LIN {X 0,Y 485.565,Z 374.75,A -85,B 0,C 180,E1 23378.433,E2 23378.433} C_VEL
LIN {X 0,Y 487.506,Z 347.224,A -85,B 0,C 180,E1 23374.747,E2 23374.747} C_VEL
LIN {X 0,Y 489.864,Z 321.169,A -85,B 0,C 180,E1 23371.121,E2 23371.121} C_VEL
LIN {X 0,Y 489.847,Z 318.644,A -85,B 0,C 180,E1 23370.733,E2 23370.733} C_VEL
LIN {X 0,Y 486.96,Z 308.048,A -85,B 0,C 180,E1 23368.702,E2 23368.702} C_VEL
LIN {X 0,Y 483.664,Z 298.045,A -85,B 0,C 180,E1 23366.497,E2 23366.497} C_VEL
LIN {X 0,Y 480.889,Z 290.899,A -85,B 0,C 180,E1 23364.593,E2 23364.593} C_VEL
LIN {X 0,Y 480.887,Z 290.899,A -85,B 0,C 180,E1 23360.949,E2 23360.949} C_VEL
LIN {X 0,Y 480.886,Z 290.899,A -85,B 0,C 180,E1 23357.325,E2 23357.325} C_VEL
LIN {X 0,Y 480.891,Z 290.899,A -85,B 0,C 180,E1 23353.65,E2 23353.65} C_VEL
LIN {X 0,Y 480.897,Z 290.898,A -85,B 0,C 180,E1 23349.976,E2 23349.976} C_VEL
LIN {X 0,Y 480.854,Z 290.925,A -85,B 0,C 180,E1 23348.951,E2 23348.951} C_VEL
LIN {X 0,Y 482.165,Z 294.329,A -85,B 0,C 180,E1 23348.168,E2 23348.168} C_VEL
LIN {X 0,Y 482.997,Z 296.239,A -85,B 0,C 180,E1 23347.74,E2 23347.74} C_VEL
LIN {X 0,Y 486.121,Z 303.618,A -85,B 0,C 180,E1 23346.266,E2 23346.266} C_VEL
LIN {X 0,Y 489.9,Z 313.848,A -85,B 0,C 180,E1 23344.569,E2 23344.569} C_VEL
LIN {X 0,Y 492.294,Z 321.57,A -85,B 0,C 180,E1 23343.465,E2 23343.465} C_VEL
LIN {X 0,Y 489.453,Z 352.379,A -85,B 0,C 180,E1 23340.575,E2 23340.575} C_VEL
LIN {X 0,Y 487.08,Z 389.197,A -85,B 0,C 180,E1 23337.373,E2 23337.373} C_VEL
LIN {X 0,Y 488.749,Z 404.821,A -85,B 0,C 180,E1 23337.007,E2 23337.007} C_VEL
LIN {X 0,Y 487.087,Z 540.591,A -85,B 0,C 180,E1 23334.828,E2 23334.828} C_VEL
LIN {X 0,Y 486.559,Z 592.008,A -85,B 0,C 180,E1 23334.024,E2 23334.024} C_VEL
LIN {X 0,Y 485.998,Z 611.058,A -85,B 0,C 180,E1 23333.512,E2 23333.512} C_VEL
LIN {X 0,Y 485.301,Z 630.353,A -85,B 0,C 180,E1 23332.758,E2 23332.758} C_VEL
LIN {X 0,Y 484.52,Z 648.608,A -85,B 0,C 180,E1 23331.806,E2 23331.806} C_VEL
LIN {X 0,Y 483.712,Z 665.393,A -85,B 0,C 180,E1 23330.7,E2 23330.7} C_VEL
LIN {X 0,Y 482.923,Z 681.405,A -85,B 0,C 180,E1 23329.41,E2 23329.41} C_VEL
LIN {X 0,Y 482.19,Z 696.517,A -85,B 0,C 180,E1 23327.935,E2 23327.935} C_VEL
LIN {X 0,Y 481.525,Z 710.621,A -85,B 0,C 180,E1 23326.28,E2 23326.28} C_VEL
LIN {X 0,Y 480.991,Z 723.539,A -85,B 0,C 180,E1 23324.446,E2 23324.446} C_VEL
LIN {X 0,Y 480.599,Z 734.198,A -85,B 0,C 180,E1 23322.619,E2 23322.619} C_VEL
LIN {X 0,Y 480.349,Z 743.484,A -85,B 0,C 180,E1 23320.677,E2 23320.677} C_VEL
LIN {X 0,Y 480.202,Z 751.314,A -85,B 0,C 180,E1 23318.623,E2 23318.623} C_VEL
LIN {X 0,Y 480.129,Z 757.3,A -85,B 0,C 180,E1 23316.578,E2 23316.578} C_VEL
LIN {X 0,Y 480.123,Z 761.787,A -85,B 0,C 180,E1 23314.42,E2 23314.42} C_VEL
LIN {X 0,Y 480.138,Z 764.484,A -85,B 0,C 180,E1 23312.268,E2 23312.268} C_VEL
LIN {X 0,Y 480.148,Z 765.458,A -85,B 0,C 180,E1 23310.12,E2 23310.12} C_VEL
LIN {X 0,Y 480.133,Z 764.739,A -85,B 0,C 180,E1 23307.972,E2 23307.972} C_VEL
LIN {X 0,Y 480.108,Z 762.322,A -85,B 0,C 180,E1 23305.821,E2 23305.821} C_VEL
LIN {X 0,Y 480.107,Z 758.423,A -85,B 0,C 180,E1 23303.784,E2 23303.784} C_VEL
LIN {X 0,Y 480.159,Z 752.88,A -85,B 0,C 180,E1 23301.74,E2 23301.74} C_VEL
LIN {X 0,Y 480.289,Z 745.557,A -85,B 0,C 180,E1 23299.688,E2 23299.688} C_VEL
LIN {X 0,Y 480.52,Z 736.848,A -85,B 0,C 180,E1 23297.747,E2 23297.747} C_VEL
LIN {X 0,Y 480.923,Z 726.12,A -85,B 0,C 180,E1 23295.8,E2 23295.8} C_VEL
LIN {X 0,Y 481.465,Z 713.873,A -85,B 0,C 180,E1 23293.967,E2 23293.967} C_VEL
LIN {X 0,Y 482.149,Z 700.593,A -85,B 0,C 180,E1 23292.315,E2 23292.315} C_VEL
LIN {X 0,Y 482.946,Z 685.825,A -85,B 0,C 180,E1 23290.782,E2 23290.782} C_VEL
LIN {X 0,Y 483.809,Z 669.989,A -85,B 0,C 180,E1 23289.422,E2 23289.422} C_VEL
LIN {X 0,Y 484.74,Z 652.554,A -85,B 0,C 180,E1 23288.206,E2 23288.206} C_VEL
LIN {X 0,Y 485.594,Z 634.78,A -85,B 0,C 180,E1 23287.227,E2 23287.227} C_VEL
LIN {X 0,Y 486.357,Z 616.371,A -85,B 0,C 180,E1 23286.454,E2 23286.454} C_VEL
LIN {X 0,Y 486.978,Z 597.757,A -85,B 0,C 180,E1 23285.901,E2 23285.901} C_VEL
LIN {X 0,Y 487.355,Z 575.191,A -85,B 0,C 180,E1 23285.49,E2 23285.49} C_VEL
LIN {X 0,Y 489.185,Z 402.332,A -85,B 0,C 180,E1 23282.787,E2 23282.787} C_VEL
LIN {X 0,Y 487.295,Z 387.28,A -85,B 0,C 180,E1 23282.426,E2 23282.426} C_VEL
LIN {X 0,Y 489.759,Z 341.908,A -85,B 0,C 180,E1 23278.629,E2 23278.629} C_VEL
LIN {X 0,Y 490.955,Z 319.92,A -85,B 0,C 180,E1 23276.733,E2 23276.733} C_VEL
LIN {X 0,Y 483.773,Z 299.432,A -85,B 0,C 180,E1 23274.317,E2 23274.317} C_VEL
LIN {X 0,Y 480.829,Z 290.905,A -85,B 0,C 180,E1 23273.249,E2 23273.249} C_VEL
LIN {X 0,Y 480.878,Z 290.9,A -85,B 0,C 180,E1 23269.738,E2 23269.738} C_VEL
LIN {X 0,Y 480.837,Z 290.903,A -85,B 0,C 180,E1 23266.178,E2 23266.178} C_VEL
LIN {X 0,Y 480.812,Z 290.901,A -85,B 0,C 180,E1 23262.683,E2 23262.683} C_VEL
LIN {X 0,Y 480.826,Z 290.901,A -85,B 0,C 180,E1 23259.139,E2 23259.139} C_VEL
LIN {X 0,Y 480.872,Z 290.901,A -85,B 0,C 180,E1 23255.753,E2 23255.753} C_VEL
LIN {X 0,Y 480.835,Z 290.9,A -85,B 0,C 180,E1 23252.164,E2 23252.164} C_VEL
LIN {X 0,Y 480.816,Z 290.9,A -85,B 0,C 180,E1 23248.711,E2 23248.711} C_VEL
LIN {X 0,Y 480.841,Z 290.899,A -85,B 0,C 180,E1 23245.233,E2 23245.233} C_VEL
LIN {X 0,Y 480.882,Z 290.9,A -85,B 0,C 180,E1 23241.723,E2 23241.723} C_VEL
LIN {X 0,Y 480.837,Z 290.9,A -85,B 0,C 180,E1 23238.145,E2 23238.145} C_VEL
LIN {X 0,Y 480.818,Z 290.9,A -85,B 0,C 180,E1 23234.698,E2 23234.698} C_VEL
LIN {X 0,Y 480.851,Z 290.899,A -85,B 0,C 180,E1 23231.273,E2 23231.273} C_VEL
LIN {X 0,Y 480.872,Z 290.9,A -85,B 0,C 180,E1 23227.769,E2 23227.769} C_VEL
LIN {X 0,Y 480.828,Z 290.899,A -85,B 0,C 180,E1 23224.295,E2 23224.295} C_VEL
LIN {X 0,Y 480.824,Z 290.899,A -85,B 0,C 180,E1 23220.717,E2 23220.717} C_VEL
LIN {X 0,Y 480.859,Z 290.898,A -85,B 0,C 180,E1 23217.261,E2 23217.261} C_VEL
LIN {X 0,Y 480.881,Z 290.9,A -85,B 0,C 180,E1 23213.641,E2 23213.641} C_VEL
LIN {X 0,Y 480.834,Z 290.899,A -85,B 0,C 180,E1 23210.184,E2 23210.184} C_VEL
LIN {X 0,Y 480.828,Z 290.898,A -85,B 0,C 180,E1 23206.657,E2 23206.657} C_VEL
LIN {X 0,Y 480.864,Z 290.897,A -85,B 0,C 180,E1 23203.203,E2 23203.203} C_VEL
LIN {X 0,Y 480.877,Z 290.9,A -85,B 0,C 180,E1 23199.672,E2 23199.672} C_VEL
LIN {X 0,Y 480.835,Z 290.899,A -85,B 0,C 180,E1 23196.211,E2 23196.211} C_VEL
LIN {X 0,Y 480.832,Z 290.898,A -85,B 0,C 180,E1 23192.61,E2 23192.61} C_VEL
LIN {X 0,Y 480.87,Z 290.896,A -85,B 0,C 180,E1 23189.173,E2 23189.173} C_VEL
LIN {X 0,Y 480.876,Z 290.9,A -85,B 0,C 180,E1 23185.633,E2 23185.633} C_VEL
LIN {X 0,Y 480.837,Z 290.898,A -85,B 0,C 180,E1 23182.165,E2 23182.165} C_VEL
LIN {X 0,Y 480.837,Z 290.897,A -85,B 0,C 180,E1 23178.608,E2 23178.608} C_VEL
LIN {X 0,Y 480.877,Z 290.896,A -85,B 0,C 180,E1 23175.154,E2 23175.154} C_VEL
LIN {X 0,Y 480.884,Z 290.9,A -85,B 0,C 180,E1 23171.542,E2 23171.542} C_VEL
LIN {X 0,Y 480.839,Z 290.898,A -85,B 0,C 180,E1 23168.138,E2 23168.138} C_VEL
LIN {X 0,Y 480.842,Z 290.897,A -85,B 0,C 180,E1 23164.574,E2 23164.574} C_VEL
LIN {X 0,Y 480.874,Z 290.895,A -85,B 0,C 180,E1 23161.04,E2 23161.04} C_VEL
LIN {X 0,Y 480.844,Z 290.898,A -85,B 0,C 180,E1 23158.07,E2 23158.07} C_VEL
LIN {X 0,Y 479.865,Z 291.024,A -85,B 0,C 180,E1 23157.151,E2 23157.151} C_VEL
LIN {X 0,Y 473.419,Z 291.823,A -85,B 0,C 180,E1 23154.569,E2 23154.569} C_VEL
LIN {X 0,Y 472.913,Z 291.887,A -85,B 0,C 180,E1 23153.895,E2 23153.895} C_VEL
LIN {X 0,Y 472.904,Z 291.885,A -85,B 0,C 180,E1 23150.416,E2 23150.416} C_VEL
LIN {X 0,Y 472.924,Z 291.884,A -85,B 0,C 180,E1 23146.836,E2 23146.836} C_VEL
LIN {X 0,Y 472.954,Z 291.886,A -85,B 0,C 180,E1 23143.322,E2 23143.322} C_VEL
LIN {X 0,Y 472.921,Z 291.888,A -85,B 0,C 180,E1 23139.737,E2 23139.737} C_VEL
LIN {X 0,Y 472.905,Z 291.886,A -85,B 0,C 180,E1 23136.189,E2 23136.189} C_VEL
LIN {X 0,Y 472.914,Z 291.884,A -85,B 0,C 180,E1 23132.544,E2 23132.544} C_VEL
LIN {X 0,Y 472.949,Z 291.883,A -85,B 0,C 180,E1 23129.03,E2 23129.03} C_VEL
LIN {X 0,Y 472.945,Z 291.889,A -85,B 0,C 180,E1 23125.391,E2 23125.391} C_VEL
LIN {X 0,Y 472.914,Z 291.887,A -85,B 0,C 180,E1 23121.856,E2 23121.856} C_VEL
LIN {X 0,Y 472.908,Z 291.885,A -85,B 0,C 180,E1 23118.197,E2 23118.197} C_VEL
LIN {X 0,Y 472.924,Z 291.883,A -85,B 0,C 180,E1 23114.585,E2 23114.585} C_VEL
LIN {X 0,Y 472.953,Z 291.883,A -85,B 0,C 180,E1 23110.999,E2 23110.999} C_VEL
LIN {X 0,Y 472.951,Z 291.888,A -85,B 0,C 180,E1 23107.37,E2 23107.37} C_VEL
LIN {X 0,Y 472.92,Z 291.886,A -85,B 0,C 180,E1 23103.776,E2 23103.776} C_VEL
LIN {X 0,Y 472.914,Z 291.884,A -85,B 0,C 180,E1 23100.207,E2 23100.207} C_VEL
LIN {X 0,Y 472.934,Z 291.883,A -85,B 0,C 180,E1 23096.62,E2 23096.62} C_VEL
LIN {X 0,Y 472.955,Z 291.883,A -85,B 0,C 180,E1 23092.949,E2 23092.949} C_VEL
LIN {X 0,Y 472.946,Z 291.888,A -85,B 0,C 180,E1 23089.369,E2 23089.369} C_VEL
LIN {X 0,Y 472.922,Z 291.886,A -85,B 0,C 180,E1 23085.757,E2 23085.757} C_VEL
LIN {X 0,Y 472.917,Z 291.884,A -85,B 0,C 180,E1 23082.08,E2 23082.08} C_VEL
LIN {X 0,Y 472.938,Z 291.885,A -85,B 0,C 180,E1 23078.533,E2 23078.533} C_VEL
LIN {X 0,Y 472.955,Z 291.885,A -85,B 0,C 180,E1 23074.888,E2 23074.888} C_VEL
LIN {X 0,Y 472.943,Z 292.039,A -85,B 0,C 180,E1 23072.224,E2 23072.224} C_VEL
LIN {X 0,Y 478.316,Z 312.031,A -85,B 0,C 180,E1 23069.098,E2 23069.098} C_VEL
LIN {X 0,Y 479.02,Z 316.059,A -85,B 0,C 180,E1 23068.506,E2 23068.506} C_VEL
LIN {X 0,Y 477.486,Z 344.796,A -85,B 0,C 180,E1 23064.756,E2 23064.756} C_VEL
LIN {X 0,Y 476.1,Z 374.187,A -85,B 0,C 180,E1 23060.979,E2 23060.979} C_VEL
LIN {X 0,Y 474.868,Z 403.252,A -85,B 0,C 180,E1 23057.3,E2 23057.3} C_VEL
LIN {X 0,Y 475.312,Z 406.497,A -85,B 0,C 180,E1 23057.183,E2 23057.183} C_VEL
LIN {X 0,Y 477.218,Z 420.131,A -85,B 0,C 180,E1 23056.849,E2 23056.849} C_VEL
LIN {X 0,Y 475.77,Z 522.315,A -85,B 0,C 180,E1 23055.029,E2 23055.029} C_VEL
LIN {X 0,Y 475.486,Z 537.221,A -85,B 0,C 180,E1 23054.552,E2 23054.552} C_VEL
LIN {X 0,Y 475.065,Z 552.814,A -85,B 0,C 180,E1 23053.803,E2 23053.803} C_VEL
LIN {X 0,Y 474.577,Z 567.324,A -85,B 0,C 180,E1 23052.84,E2 23052.84} C_VEL
LIN {X 0,Y 474.106,Z 579.994,A -85,B 0,C 180,E1 23051.74,E2 23051.74} C_VEL
LIN {X 0,Y 473.699,Z 590.671,A -85,B 0,C 180,E1 23050.58,E2 23050.58} C_VEL
LIN {X 0,Y 473.281,Z 601.28,A -85,B 0,C 180,E1 23049.115,E2 23049.115} C_VEL
LIN {X 0,Y 472.98,Z 609.588,A -85,B 0,C 180,E1 23047.651,E2 23047.651} C_VEL
LIN {X 0,Y 472.774,Z 616.567,A -85,B 0,C 180,E1 23046.068,E2 23046.068} C_VEL
LIN {X 0,Y 472.634,Z 622.024,A -85,B 0,C 180,E1 23044.366,E2 23044.366} C_VEL
LIN {X 0,Y 472.574,Z 625.726,A -85,B 0,C 180,E1 23042.666,E2 23042.666} C_VEL
LIN {X 0,Y 472.57,Z 627.887,A -85,B 0,C 180,E1 23040.726,E2 23040.726} C_VEL
LIN {X 0,Y 472.607,Z 627.981,A -85,B 0,C 180,E1 23038.907,E2 23038.907} C_VEL
LIN {X 0,Y 472.689,Z 626.442,A -85,B 0,C 180,E1 23037.21,E2 23037.21} C_VEL
LIN {X 0,Y 472.836,Z 622.885,A -85,B 0,C 180,E1 23035.389,E2 23035.389} C_VEL
LIN {X 0,Y 473.043,Z 617.692,A -85,B 0,C 180,E1 23033.688,E2 23033.688} C_VEL
LIN {X 0,Y 473.336,Z 611.053,A -85,B 0,C 180,E1 23032.107,E2 23032.107} C_VEL
LIN {X 0,Y 473.736,Z 602.21,A -85,B 0,C 180,E1 23030.523,E2 23030.523} C_VEL
LIN {X 0,Y 474.207,Z 592.121,A -85,B 0,C 180,E1 23029.121,E2 23029.121} C_VEL
LIN {X 0,Y 474.72,Z 580.397,A -85,B 0,C 180,E1 23027.84,E2 23027.84} C_VEL
LIN {X 0,Y 475.257,Z 567.484,A -85,B 0,C 180,E1 23026.742,E2 23026.742} C_VEL
LIN {X 0,Y 475.754,Z 553.464,A -85,B 0,C 180,E1 23025.826,E2 23025.826} C_VEL
LIN {X 0,Y 476.183,Z 539.021,A -85,B 0,C 180,E1 23025.125,E2 23025.125} C_VEL
LIN {X 0,Y 476.527,Z 523.033,A -85,B 0,C 180,E1 23024.595,E2 23024.595} C_VEL
LIN {X 0,Y 479.34,Z 425.993,A -85,B 0,C 180,E1 23022.487,E2 23022.487} C_VEL
LIN {X 0,Y 479.361,Z 419.035,A -85,B 0,C 180,E1 23022.314,E2 23022.314} C_VEL
LIN {X 0,Y 476.547,Z 403.549,A -85,B 0,C 180,E1 23021.718,E2 23021.718} C_VEL
LIN {X 0,Y 478.233,Z 375.694,A -85,B 0,C 180,E1 23018.021,E2 23018.021} C_VEL
LIN {X 0,Y 480.426,Z 347.936,A -85,B 0,C 180,E1 23014.215,E2 23014.215} C_VEL
LIN {X 0,Y 483.024,Z 322.741,A -85,B 0,C 180,E1 23010.619,E2 23010.619} C_VEL
LIN {X 0,Y 480.339,Z 312.444,A -85,B 0,C 180,E1 23008.589,E2 23008.589} C_VEL
LIN {X 0,Y 477.229,Z 302.718,A -85,B 0,C 180,E1 23006.366,E2 23006.366} C_VEL
LIN {X 0,Y 474.194,Z 295.278,A -85,B 0,C 180,E1 23004.262,E2 23004.262} C_VEL
LIN {X 0,Y 472.951,Z 291.888,A -85,B 0,C 180,E1 23003.1,E2 23003.1} C_VEL
LIN {X 0,Y 472.948,Z 291.888,A -85,B 0,C 180,E1 22999.53,E2 22999.53} C_VEL
LIN {X 0,Y 472.952,Z 291.887,A -85,B 0,C 180,E1 22995.929,E2 22995.929} C_VEL
LIN {X 0,Y 472.952,Z 291.888,A -85,B 0,C 180,E1 22992.244,E2 22992.244} C_VEL
LIN {X 0,Y 472.953,Z 291.966,A -85,B 0,C 180,E1 22990.361,E2 22990.361} C_VEL
LIN {X 0,Y 474.397,Z 295.616,A -85,B 0,C 180,E1 22989.329,E2 22989.329} C_VEL
LIN {X 0,Y 476.868,Z 301.021,A -85,B 0,C 180,E1 22987.966,E2 22987.966} C_VEL
LIN {X 0,Y 480.14,Z 309.138,A -85,B 0,C 180,E1 22986.302,E2 22986.302} C_VEL
LIN {X 0,Y 483.603,Z 319.023,A -85,B 0,C 180,E1 22984.625,E2 22984.625} C_VEL
LIN {X 0,Y 485.319,Z 325.278,A -85,B 0,C 180,E1 22983.727,E2 22983.727} C_VEL
LIN {X 0,Y 482.178,Z 355.567,A -85,B 0,C 180,E1 22980.81,E2 22980.81} C_VEL
LIN {X 0,Y 479.741,Z 389.652,A -85,B 0,C 180,E1 22977.775,E2 22977.775} C_VEL
LIN {X 0,Y 481.429,Z 405.855,A -85,B 0,C 180,E1 22977.377,E2 22977.377} C_VEL
LIN {X 0,Y 479.592,Z 536.545,A -85,B 0,C 180,E1 22975.211,E2 22975.211} C_VEL
LIN {X 0,Y 478.968,Z 591.308,A -85,B 0,C 180,E1 22974.334,E2 22974.334} C_VEL
LIN {X 0,Y 478.366,Z 610.338,A -85,B 0,C 180,E1 22973.812,E2 22973.812} C_VEL
LIN {X 0,Y 477.612,Z 629.542,A -85,B 0,C 180,E1 22973.047,E2 22973.047} C_VEL
LIN {X 0,Y 476.794,Z 647.206,A -85,B 0,C 180,E1 22972.113,E2 22972.113} C_VEL
LIN {X 0,Y 475.924,Z 664.054,A -85,B 0,C 180,E1 22970.991,E2 22970.991} C_VEL
LIN {X 0,Y 475.077,Z 680.111,A -85,B 0,C 180,E1 22969.679,E2 22969.679} C_VEL
LIN {X 0,Y 474.297,Z 695.261,A -85,B 0,C 180,E1 22968.18,E2 22968.18} C_VEL
LIN {X 0,Y 473.592,Z 709.421,A -85,B 0,C 180,E1 22966.498,E2 22966.498} C_VEL
LIN {X 0,Y 473.051,Z 722.005,A -85,B 0,C 180,E1 22964.694,E2 22964.694} C_VEL
LIN {X 0,Y 472.625,Z 733.381,A -85,B 0,C 180,E1 22962.711,E2 22962.711} C_VEL
LIN {X 0,Y 472.375,Z 742.63,A -85,B 0,C 180,E1 22960.736,E2 22960.736} C_VEL
LIN {X 0,Y 472.239,Z 750.419,A -85,B 0,C 180,E1 22958.647,E2 22958.647} C_VEL
LIN {X 0,Y 472.182,Z 756.367,A -85,B 0,C 180,E1 22956.567,E2 22956.567} C_VEL
LIN {X 0,Y 472.191,Z 760.8,A -85,B 0,C 180,E1 22954.373,E2 22954.373} C_VEL
LIN {X 0,Y 472.217,Z 763.445,A -85,B 0,C 180,E1 22952.185,E2 22952.185} C_VEL
LIN {X 0,Y 472.229,Z 764.363,A -85,B 0,C 180,E1 22950.001,E2 22950.001} C_VEL
LIN {X 0,Y 472.2,Z 763.565,A -85,B 0,C 180,E1 22947.817,E2 22947.817} C_VEL
LIN {X 0,Y 472.161,Z 761.049,A -85,B 0,C 180,E1 22945.629,E2 22945.629} C_VEL
LIN {X 0,Y 472.143,Z 756.768,A -85,B 0,C 180,E1 22943.434,E2 22943.434} C_VEL
LIN {X 0,Y 472.198,Z 750.616,A -85,B 0,C 180,E1 22941.232,E2 22941.232} C_VEL
LIN {X 0,Y 472.345,Z 742.923,A -85,B 0,C 180,E1 22939.142,E2 22939.142} C_VEL
LIN {X 0,Y 472.647,Z 733.161,A -85,B 0,C 180,E1 22937.043,E2 22937.043} C_VEL
LIN {X 0,Y 473.084,Z 722.591,A -85,B 0,C 180,E1 22935.184,E2 22935.184} C_VEL
LIN {X 0,Y 473.706,Z 709.753,A -85,B 0,C 180,E1 22933.319,E2 22933.319} C_VEL
LIN {X 0,Y 474.482,Z 695.805,A -85,B 0,C 180,E1 22931.638,E2 22931.638} C_VEL
LIN {X 0,Y 475.345,Z 680.801,A -85,B 0,C 180,E1 22930.136,E2 22930.136} C_VEL
LIN {X 0,Y 476.327,Z 663.906,A -85,B 0,C 180,E1 22928.75,E2 22928.75} C_VEL
LIN {X 0,Y 477.249,Z 647.358,A -85,B 0,C 180,E1 22927.652,E2 22927.652} C_VEL
LIN {X 0,Y 478.137,Z 629.658,A -85,B 0,C 180,E1 22926.721,E2 22926.721} C_VEL
LIN {X 0,Y 478.905,Z 611.189,A -85,B 0,C 180,E1 22925.989,E2 22925.989} C_VEL
LIN {X 0,Y 479.525,Z 592.27,A -85,B 0,C 180,E1 22925.474,E2 22925.474} C_VEL
LIN {X 0,Y 481.747,Z 402.99,A -85,B 0,C 180,E1 22922.428,E2 22922.428} C_VEL
LIN {X 0,Y 479.824,Z 387.274,A -85,B 0,C 180,E1 22922.041,E2 22922.041} C_VEL
LIN {X 0,Y 482.517,Z 341.869,A -85,B 0,C 180,E1 22918.168,E2 22918.168} C_VEL
LIN {X 0,Y 483.699,Z 322.82,A -85,B 0,C 180,E1 22916.503,E2 22916.503} C_VEL
LIN {X 0,Y 475.815,Z 300.286,A -85,B 0,C 180,E1 22913.797,E2 22913.797} C_VEL
LIN {X 0,Y 472.876,Z 291.895,A -85,B 0,C 180,E1 22912.716,E2 22912.716} C_VEL
LIN {X 0,Y 472.887,Z 291.894,A -85,B 0,C 180,E1 22909.197,E2 22909.197} C_VEL
LIN {X 0,Y 472.929,Z 291.889,A -85,B 0,C 180,E1 22905.76,E2 22905.76} C_VEL
LIN {X 0,Y 472.891,Z 291.89,A -85,B 0,C 180,E1 22902.251,E2 22902.251} C_VEL
LIN {X 0,Y 472.874,Z 291.889,A -85,B 0,C 180,E1 22898.721,E2 22898.721} C_VEL
LIN {X 0,Y 472.898,Z 291.889,A -85,B 0,C 180,E1 22895.256,E2 22895.256} C_VEL
LIN {X 0,Y 472.933,Z 291.889,A -85,B 0,C 180,E1 22891.623,E2 22891.623} C_VEL
LIN {X 0,Y 472.899,Z 291.889,A -85,B 0,C 180,E1 22888.133,E2 22888.133} C_VEL
LIN {X 0,Y 472.88,Z 291.889,A -85,B 0,C 180,E1 22884.609,E2 22884.609} C_VEL
LIN {X 0,Y 472.891,Z 291.888,A -85,B 0,C 180,E1 22881.067,E2 22881.067} C_VEL
LIN {X 0,Y 472.934,Z 291.888,A -85,B 0,C 180,E1 22877.548,E2 22877.548} C_VEL
LIN {X 0,Y 472.915,Z 291.889,A -85,B 0,C 180,E1 22873.948,E2 22873.948} C_VEL
LIN {X 0,Y 472.884,Z 291.888,A -85,B 0,C 180,E1 22870.478,E2 22870.478} C_VEL
LIN {X 0,Y 472.886,Z 291.888,A -85,B 0,C 180,E1 22866.802,E2 22866.802} C_VEL
LIN {X 0,Y 472.917,Z 291.887,A -85,B 0,C 180,E1 22863.274,E2 22863.274} C_VEL
LIN {X 0,Y 472.946,Z 291.889,A -85,B 0,C 180,E1 22859.638,E2 22859.638} C_VEL
LIN {X 0,Y 472.9,Z 291.888,A -85,B 0,C 180,E1 22856.122,E2 22856.122} C_VEL
LIN {X 0,Y 472.887,Z 291.888,A -85,B 0,C 180,E1 22852.577,E2 22852.577} C_VEL
LIN {X 0,Y 472.905,Z 291.887,A -85,B 0,C 180,E1 22849.033,E2 22849.033} C_VEL
LIN {X 0,Y 472.949,Z 291.886,A -85,B 0,C 180,E1 22845.431,E2 22845.431} C_VEL
LIN {X 0,Y 472.926,Z 291.889,A -85,B 0,C 180,E1 22841.768,E2 22841.768} C_VEL
LIN {X 0,Y 472.893,Z 291.888,A -85,B 0,C 180,E1 22838.286,E2 22838.286} C_VEL
LIN {X 0,Y 472.892,Z 291.887,A -85,B 0,C 180,E1 22834.585,E2 22834.585} C_VEL
LIN {X 0,Y 472.917,Z 291.886,A -85,B 0,C 180,E1 22831.045,E2 22831.045} C_VEL
LIN {X 0,Y 472.946,Z 291.888,A -85,B 0,C 180,E1 22827.512,E2 22827.512} C_VEL
LIN {X 0,Y 472.906,Z 291.888,A -85,B 0,C 180,E1 22824.004,E2 22824.004} C_VEL
LIN {X 0,Y 472.894,Z 291.887,A -85,B 0,C 180,E1 22820.478,E2 22820.478} C_VEL
LIN {X 0,Y 472.922,Z 291.885,A -85,B 0,C 180,E1 22817.012,E2 22817.012} C_VEL
LIN {X 0,Y 472.947,Z 291.887,A -85,B 0,C 180,E1 22813.398,E2 22813.398} C_VEL
LIN {X 0,Y 472.917,Z 291.888,A -85,B 0,C 180,E1 22809.836,E2 22809.836} C_VEL
LIN {X 0,Y 472.899,Z 291.886,A -85,B 0,C 180,E1 22806.298,E2 22806.298} C_VEL
LIN {X 0,Y 472.906,Z 291.885,A -85,B 0,C 180,E1 22802.624,E2 22802.624} C_VEL
LIN {X 0,Y 472.943,Z 291.884,A -85,B 0,C 180,E1 22799.093,E2 22799.093} C_VEL
LIN {X 0,Y 472.945,Z 291.889,A -85,B 0,C 180,E1 22795.488,E2 22795.488} C_VEL
LIN {X 0,Y 472.913,Z 291.887,A -85,B 0,C 180,E1 22793.895,E2 22793.895} C_VEL
LIN {X 0,Y 471.945,Z 292.013,A -85,B 0,C 180,E1 22792.962,E2 22792.962} C_VEL
LIN {X 0,Y 465.485,Z 292.81,A -85,B 0,C 180,E1 22790.336,E2 22790.336} C_VEL
LIN {X 0,Y 464.992,Z 292.877,A -85,B 0,C 180,E1 22789.65,E2 22789.65} C_VEL
LIN {X 0,Y 464.966,Z 292.875,A -85,B 0,C 180,E1 22786.104,E2 22786.104} C_VEL
LIN {X 0,Y 464.967,Z 292.874,A -85,B 0,C 180,E1 22782.417,E2 22782.417} C_VEL
LIN {X 0,Y 464.995,Z 292.873,A -85,B 0,C 180,E1 22778.905,E2 22778.905} C_VEL
LIN {X 0,Y 465.014,Z 292.875,A -85,B 0,C 180,E1 22775.304,E2 22775.304} C_VEL
LIN {X 0,Y 464.993,Z 292.877,A -85,B 0,C 180,E1 22771.601,E2 22771.601} C_VEL
LIN {X 0,Y 464.969,Z 292.875,A -85,B 0,C 180,E1 22768.027,E2 22768.027} C_VEL
LIN {X 0,Y 464.969,Z 292.874,A -85,B 0,C 180,E1 22764.322,E2 22764.322} C_VEL
LIN {X 0,Y 465.001,Z 292.872,A -85,B 0,C 180,E1 22760.843,E2 22760.843} C_VEL
LIN {X 0,Y 465.016,Z 292.874,A -85,B 0,C 180,E1 22757.204,E2 22757.204} C_VEL
LIN {X 0,Y 464.989,Z 292.876,A -85,B 0,C 180,E1 22753.638,E2 22753.638} C_VEL
LIN {X 0,Y 464.974,Z 292.874,A -85,B 0,C 180,E1 22749.993,E2 22749.993} C_VEL
LIN {X 0,Y 464.977,Z 292.873,A -85,B 0,C 180,E1 22746.289,E2 22746.289} C_VEL
LIN {X 0,Y 465.003,Z 292.871,A -85,B 0,C 180,E1 22742.741,E2 22742.741} C_VEL
LIN {X 0,Y 465.019,Z 292.873,A -85,B 0,C 180,E1 22739.076,E2 22739.076} C_VEL
LIN {X 0,Y 465.004,Z 292.877,A -85,B 0,C 180,E1 22735.412,E2 22735.412} C_VEL
LIN {X 0,Y 464.978,Z 292.874,A -85,B 0,C 180,E1 22731.891,E2 22731.891} C_VEL
LIN {X 0,Y 464.979,Z 292.873,A -85,B 0,C 180,E1 22728.194,E2 22728.194} C_VEL
LIN {X 0,Y 465.002,Z 292.872,A -85,B 0,C 180,E1 22724.624,E2 22724.624} C_VEL
LIN {X 0,Y 465.021,Z 292.873,A -85,B 0,C 180,E1 22720.976,E2 22720.976} C_VEL
LIN {X 0,Y 465.007,Z 292.878,A -85,B 0,C 180,E1 22717.289,E2 22717.289} C_VEL
LIN {X 0,Y 464.986,Z 292.878,A -85,B 0,C 180,E1 22713.677,E2 22713.677} C_VEL
LIN {X 0,Y 465.03,Z 293.02,A -85,B 0,C 180,E1 22712.658,E2 22712.658} C_VEL
LIN {X 0,Y 470.563,Z 313.554,A -85,B 0,C 180,E1 22709.393,E2 22709.393} C_VEL
LIN {X 0,Y 471.46,Z 318.133,A -85,B 0,C 180,E1 22708.706,E2 22708.706} C_VEL
LIN {X 0,Y 469.842,Z 346.416,A -85,B 0,C 180,E1 22704.964,E2 22704.964} C_VEL
LIN {X 0,Y 468.36,Z 376.105,A -85,B 0,C 180,E1 22701.105,E2 22701.105} C_VEL
LIN {X 0,Y 467.152,Z 403.75,A -85,B 0,C 180,E1 22697.587,E2 22697.587} C_VEL
LIN {X 0,Y 469.64,Z 420.948,A -85,B 0,C 180,E1 22697.151,E2 22697.151} C_VEL
LIN {X 0,Y 468.063,Z 522.866,A -85,B 0,C 180,E1 22695.283,E2 22695.283} C_VEL
LIN {X 0,Y 467.764,Z 537.758,A -85,B 0,C 180,E1 22694.797,E2 22694.797} C_VEL
LIN {X 0,Y 467.326,Z 553.152,A -85,B 0,C 180,E1 22694.05,E2 22694.05} C_VEL
LIN {X 0,Y 466.834,Z 567.121,A -85,B 0,C 180,E1 22693.12,E2 22693.12} C_VEL
LIN {X 0,Y 466.353,Z 579.443,A -85,B 0,C 180,E1 22692.064,E2 22692.064} C_VEL
LIN {X 0,Y 465.868,Z 591.439,A -85,B 0,C 180,E1 22690.759,E2 22690.759} C_VEL
LIN {X 0,Y 465.423,Z 602.129,A -85,B 0,C 180,E1 22689.27,E2 22689.27} C_VEL
LIN {X 0,Y 465.101,Z 610.51,A -85,B 0,C 180,E1 22687.782,E2 22687.782} C_VEL
LIN {X 0,Y 464.876,Z 617.553,A -85,B 0,C 180,E1 22686.172,E2 22686.172} C_VEL
LIN {X 0,Y 464.726,Z 623.083,A -85,B 0,C 180,E1 22684.44,E2 22684.44} C_VEL
LIN {X 0,Y 464.659,Z 626.834,A -85,B 0,C 180,E1 22682.712,E2 22682.712} C_VEL
LIN {X 0,Y 464.656,Z 629.048,A -85,B 0,C 180,E1 22680.738,E2 22680.738} C_VEL
LIN {X 0,Y 464.699,Z 629.187,A -85,B 0,C 180,E1 22678.889,E2 22678.889} C_VEL
LIN {X 0,Y 464.796,Z 627.688,A -85,B 0,C 180,E1 22677.162,E2 22677.162} C_VEL
LIN {X 0,Y 464.964,Z 624.168,A -85,B 0,C 180,E1 22675.311,E2 22675.311} C_VEL
LIN {X 0,Y 465.198,Z 619,A -85,B 0,C 180,E1 22673.581,E2 22673.581} C_VEL
LIN {X 0,Y 465.527,Z 612.261,A -85,B 0,C 180,E1 22671.95,E2 22671.95} C_VEL
LIN {X 0,Y 465.956,Z 603.535,A -85,B 0,C 180,E1 22670.363,E2 22670.363} C_VEL
LIN {X 0,Y 466.467,Z 593.484,A -85,B 0,C 180,E1 22668.938,E2 22668.938} C_VEL
LIN {X 0,Y 467.029,Z 581.875,A -85,B 0,C 180,E1 22667.636,E2 22667.636} C_VEL
LIN {X 0,Y 467.646,Z 568.326,A -85,B 0,C 180,E1 22666.459,E2 22666.459} C_VEL
LIN {X 0,Y 468.182,Z 554.281,A -85,B 0,C 180,E1 22665.529,E2 22665.529} C_VEL
LIN {X 0,Y 468.639,Z 539.821,A -85,B 0,C 180,E1 22664.816,E2 22664.816} C_VEL
LIN {X 0,Y 469.007,Z 523.992,A -85,B 0,C 180,E1 22664.278,E2 22664.278} C_VEL
LIN {X 0,Y 472.168,Z 427.124,A -85,B 0,C 180,E1 22662.073,E2 22662.073} C_VEL
LIN {X 0,Y 472.177,Z 420.214,A -85,B 0,C 180,E1 22661.897,E2 22661.897} C_VEL
LIN {X 0,Y 469.151,Z 403.57,A -85,B 0,C 180,E1 22661.226,E2 22661.226} C_VEL
LIN {X 0,Y 471.005,Z 376.337,A -85,B 0,C 180,E1 22657.534,E2 22657.534} C_VEL
LIN {X 0,Y 473.431,Z 348.791,A -85,B 0,C 180,E1 22653.671,E2 22653.671} C_VEL
LIN {X 0,Y 476.047,Z 326.1,A -85,B 0,C 180,E1 22650.354,E2 22650.354} C_VEL
LIN {X 0,Y 473.482,Z 315.966,A -85,B 0,C 180,E1 22648.276,E2 22648.276} C_VEL
LIN {X 0,Y 470.7,Z 307.172,A -85,B 0,C 180,E1 22646.158,E2 22646.158} C_VEL
LIN {X 0,Y 468.123,Z 300.447,A -85,B 0,C 180,E1 22644.179,E2 22644.179} C_VEL
LIN {X 0,Y 466.511,Z 296.638,A -85,B 0,C 180,E1 22642.813,E2 22642.813} C_VEL
LIN {X 0,Y 465.014,Z 292.877,A -85,B 0,C 180,E1 22641.107,E2 22641.107} C_VEL
LIN {X 0,Y 465.011,Z 292.876,A -85,B 0,C 180,E1 22637.365,E2 22637.365} C_VEL
LIN {X 0,Y 465.013,Z 292.876,A -85,B 0,C 180,E1 22633.647,E2 22633.647} C_VEL
LIN {X 0,Y 465.038,Z 293.08,A -85,B 0,C 180,E1 22632.298,E2 22632.298} C_VEL
LIN {X 0,Y 466.632,Z 296.833,A -85,B 0,C 180,E1 22630.809,E2 22630.809} C_VEL
LIN {X 0,Y 467.307,Z 297.938,A -85,B 0,C 180,E1 22630.384,E2 22630.384} C_VEL
LIN {X 0,Y 469.416,Z 302.984,A -85,B 0,C 180,E1 22628.93,E2 22628.93} C_VEL
LIN {X 0,Y 471.234,Z 307.276,A -85,B 0,C 180,E1 22627.878,E2 22627.878} C_VEL
LIN {X 0,Y 474.461,Z 315.435,A -85,B 0,C 180,E1 22626.184,E2 22626.184} C_VEL
LIN {X 0,Y 477.806,Z 325.707,A -85,B 0,C 180,E1 22624.463,E2 22624.463} C_VEL
LIN {X 0,Y 478.435,Z 328.468,A -85,B 0,C 180,E1 22624.062,E2 22624.062} C_VEL
LIN {X 0,Y 474.874,Z 359.515,A -85,B 0,C 180,E1 22620.992,E2 22620.992} C_VEL
LIN {X 0,Y 472.459,Z 390.018,A -85,B 0,C 180,E1 22618.205,E2 22618.205} C_VEL
LIN {X 0,Y 474.18,Z 406.912,A -85,B 0,C 180,E1 22617.772,E2 22617.772} C_VEL
LIN {X 0,Y 472.145,Z 533.129,A -85,B 0,C 180,E1 22615.607,E2 22615.607} C_VEL
LIN {X 0,Y 471.416,Z 590.608,A -85,B 0,C 180,E1 22614.662,E2 22614.662} C_VEL
LIN {X 0,Y 470.762,Z 609.745,A -85,B 0,C 180,E1 22614.125,E2 22614.125} C_VEL
LIN {X 0,Y 469.958,Z 628.576,A -85,B 0,C 180,E1 22613.361,E2 22613.361} C_VEL
LIN {X 0,Y 469.086,Z 645.93,A -85,B 0,C 180,E1 22612.43,E2 22612.43} C_VEL
LIN {X 0,Y 468.158,Z 662.811,A -85,B 0,C 180,E1 22611.29,E2 22611.29} C_VEL
LIN {X 0,Y 467.241,Z 679.085,A -85,B 0,C 180,E1 22609.94,E2 22609.94} C_VEL
LIN {X 0,Y 466.386,Z 694.66,A -85,B 0,C 180,E1 22608.37,E2 22608.37} C_VEL
LIN {X 0,Y 465.667,Z 708.249,A -85,B 0,C 180,E1 22606.722,E2 22606.722} C_VEL
LIN {X 0,Y 465.077,Z 721.237,A -85,B 0,C 180,E1 22604.824,E2 22604.824} C_VEL
LIN {X 0,Y 464.664,Z 732.125,A -85,B 0,C 180,E1 22602.898,E2 22602.898} C_VEL
LIN {X 0,Y 464.4,Z 741.785,A -85,B 0,C 180,E1 22600.797,E2 22600.797} C_VEL
LIN {X 0,Y 464.277,Z 749.531,A -85,B 0,C 180,E1 22598.671,E2 22598.671} C_VEL
LIN {X 0,Y 464.237,Z 755.426,A -85,B 0,C 180,E1 22596.555,E2 22596.555} C_VEL
LIN {X 0,Y 464.257,Z 759.633,A -85,B 0,C 180,E1 22594.448,E2 22594.448} C_VEL
LIN {X 0,Y 464.29,Z 762.31,A -85,B 0,C 180,E1 22592.222,E2 22592.222} C_VEL
LIN {X 0,Y 464.307,Z 763.249,A -85,B 0,C 180,E1 22590.001,E2 22590.001} C_VEL
LIN {X 0,Y 464.27,Z 762.46,A -85,B 0,C 180,E1 22587.779,E2 22587.779} C_VEL
LIN {X 0,Y 464.22,Z 759.941,A -85,B 0,C 180,E1 22585.554,E2 22585.554} C_VEL
LIN {X 0,Y 464.187,Z 755.645,A -85,B 0,C 180,E1 22583.321,E2 22583.321} C_VEL
LIN {X 0,Y 464.233,Z 749.459,A -85,B 0,C 180,E1 22581.08,E2 22581.08} C_VEL
LIN {X 0,Y 464.374,Z 741.725,A -85,B 0,C 180,E1 22578.953,E2 22578.953} C_VEL
LIN {X 0,Y 464.665,Z 732.571,A -85,B 0,C 180,E1 22576.943,E2 22576.943} C_VEL
LIN {X 0,Y 465.147,Z 721.272,A -85,B 0,C 180,E1 22574.925,E2 22574.925} C_VEL
LIN {X 0,Y 465.769,Z 709.302,A -85,B 0,C 180,E1 22573.155,E2 22573.155} C_VEL
LIN {X 0,Y 466.586,Z 695.416,A -85,B 0,C 180,E1 22571.446,E2 22571.446} C_VEL
LIN {X 0,Y 467.492,Z 680.555,A -85,B 0,C 180,E1 22569.925,E2 22569.925} C_VEL
LIN {X 0,Y 468.468,Z 664.833,A -85,B 0,C 180,E1 22568.596,E2 22568.596} C_VEL
LIN {X 0,Y 469.451,Z 648.309,A -85,B 0,C 180,E1 22567.458,E2 22567.458} C_VEL
LIN {X 0,Y 470.447,Z 629.71,A -85,B 0,C 180,E1 22566.45,E2 22566.45} C_VEL
LIN {X 0,Y 471.273,Z 611.129,A -85,B 0,C 180,E1 22565.696,E2 22565.696} C_VEL
LIN {X 0,Y 471.932,Z 592.308,A -85,B 0,C 180,E1 22565.169,E2 22565.169} C_VEL
LIN {X 0,Y 472.679,Z 535.343,A -85,B 0,C 180,E1 22564.235,E2 22564.235} C_VEL
LIN {X 0,Y 474.332,Z 403.807,A -85,B 0,C 180,E1 22562.07,E2 22562.07} C_VEL
LIN {X 0,Y 472.353,Z 387.421,A -85,B 0,C 180,E1 22561.662,E2 22561.662} C_VEL
LIN {X 0,Y 475.308,Z 340.981,A -85,B 0,C 180,E1 22557.632,E2 22557.632} C_VEL
LIN {X 0,Y 476.236,Z 325.033,A -85,B 0,C 180,E1 22556.196,E2 22556.196} C_VEL
LIN {X 0,Y 468.071,Z 301.712,A -85,B 0,C 180,E1 22553.334,E2 22553.334} C_VEL
LIN {X 0,Y 464.963,Z 292.882,A -85,B 0,C 180,E1 22552.165,E2 22552.165} C_VEL
LIN {X 0,Y 464.937,Z 292.883,A -85,B 0,C 180,E1 22548.638,E2 22548.638} C_VEL
LIN {X 0,Y 464.939,Z 292.881,A -85,B 0,C 180,E1 22544.968,E2 22544.968} C_VEL
LIN {X 0,Y 464.974,Z 292.88,A -85,B 0,C 180,E1 22541.477,E2 22541.477} C_VEL
LIN {X 0,Y 464.983,Z 292.878,A -85,B 0,C 180,E1 22537.894,E2 22537.894} C_VEL
LIN {X 0,Y 464.95,Z 292.878,A -85,B 0,C 180,E1 22534.294,E2 22534.294} C_VEL
LIN {X 0,Y 464.938,Z 292.878,A -85,B 0,C 180,E1 22530.662,E2 22530.662} C_VEL
LIN {X 0,Y 464.95,Z 292.878,A -85,B 0,C 180,E1 22527.093,E2 22527.093} C_VEL
LIN {X 0,Y 464.995,Z 292.878,A -85,B 0,C 180,E1 22523.576,E2 22523.576} C_VEL
LIN {X 0,Y 464.971,Z 292.878,A -85,B 0,C 180,E1 22519.995,E2 22519.995} C_VEL
LIN {X 0,Y 464.944,Z 292.878,A -85,B 0,C 180,E1 22516.444,E2 22516.444} C_VEL
LIN {X 0,Y 464.944,Z 292.877,A -85,B 0,C 180,E1 22512.799,E2 22512.799} C_VEL
LIN {X 0,Y 464.973,Z 292.877,A -85,B 0,C 180,E1 22509.251,E2 22509.251} C_VEL
LIN {X 0,Y 464.999,Z 292.879,A -85,B 0,C 180,E1 22505.678,E2 22505.678} C_VEL
LIN {X 0,Y 464.961,Z 292.878,A -85,B 0,C 180,E1 22502.097,E2 22502.097} C_VEL
LIN {X 0,Y 464.946,Z 292.877,A -85,B 0,C 180,E1 22498.646,E2 22498.646} C_VEL
LIN {X 0,Y 464.966,Z 292.876,A -85,B 0,C 180,E1 22495.067,E2 22495.067} C_VEL
LIN {X 0,Y 465.005,Z 292.876,A -85,B 0,C 180,E1 22491.47,E2 22491.47} C_VEL
LIN {X 0,Y 464.982,Z 292.878,A -85,B 0,C 180,E1 22487.837,E2 22487.837} C_VEL
LIN {X 0,Y 464.951,Z 292.876,A -85,B 0,C 180,E1 22484.409,E2 22484.409} C_VEL
LIN {X 0,Y 464.956,Z 292.876,A -85,B 0,C 180,E1 22480.738,E2 22480.738} C_VEL
LIN {X 0,Y 464.993,Z 292.875,A -85,B 0,C 180,E1 22477.232,E2 22477.232} C_VEL
LIN {X 0,Y 465.002,Z 292.879,A -85,B 0,C 180,E1 22473.573,E2 22473.573} C_VEL
LIN {X 0,Y 464.964,Z 292.877,A -85,B 0,C 180,E1 22470.065,E2 22470.065} C_VEL
LIN {X 0,Y 464.955,Z 292.876,A -85,B 0,C 180,E1 22466.453,E2 22466.453} C_VEL
LIN {X 0,Y 464.968,Z 292.875,A -85,B 0,C 180,E1 22462.828,E2 22462.828} C_VEL
LIN {X 0,Y 465.018,Z 292.874,A -85,B 0,C 180,E1 22459.349,E2 22459.349} C_VEL
LIN {X 0,Y 464.992,Z 292.878,A -85,B 0,C 180,E1 22455.67,E2 22455.67} C_VEL
LIN {X 0,Y 464.964,Z 292.876,A -85,B 0,C 180,E1 22452.112,E2 22452.112} C_VEL
LIN {X 0,Y 464.96,Z 292.875,A -85,B 0,C 180,E1 22448.422,E2 22448.422} C_VEL
LIN {X 0,Y 464.982,Z 292.874,A -85,B 0,C 180,E1 22444.887,E2 22444.887} C_VEL
LIN {X 0,Y 465.017,Z 292.875,A -85,B 0,C 180,E1 22441.354,E2 22441.354} C_VEL
LIN {X 0,Y 464.98,Z 292.876,A -85,B 0,C 180,E1 22437.814,E2 22437.814} C_VEL
LIN {X 0,Y 464.964,Z 292.875,A -85,B 0,C 180,E1 22434.249,E2 22434.249} C_VEL
LIN {X 0,Y 464.973,Z 292.874,A -85,B 0,C 180,E1 22430.649,E2 22430.649} C_VEL
LIN {X 0,Y 464.992,Z 292.877,A -85,B 0,C 180,E1 22429.65,E2 22429.65} C_VEL
LIN {X 0,Y 464.051,Z 293.006,A -85,B 0,C 180,E1 22428.701,E2 22428.701} C_VEL
LIN {X 0,Y 457.498,Z 293.82,A -85,B 0,C 180,E1 22425.962,E2 22425.962} C_VEL
LIN {X 0,Y 457.077,Z 293.864,A -85,B 0,C 180,E1 22425.334,E2 22425.334} C_VEL
LIN {X 0,Y 457.045,Z 293.865,A -85,B 0,C 180,E1 22421.738,E2 22421.738} C_VEL
LIN {X 0,Y 457.026,Z 293.864,A -85,B 0,C 180,E1 22418.174,E2 22418.174} C_VEL
LIN {X 0,Y 457.033,Z 293.863,A -85,B 0,C 180,E1 22414.516,E2 22414.516} C_VEL
LIN {X 0,Y 457.06,Z 293.861,A -85,B 0,C 180,E1 22410.876,E2 22410.876} C_VEL
LIN {X 0,Y 457.074,Z 293.864,A -85,B 0,C 180,E1 22407.241,E2 22407.241} C_VEL
LIN {X 0,Y 457.055,Z 293.865,A -85,B 0,C 180,E1 22403.593,E2 22403.593} C_VEL
LIN {X 0,Y 457.033,Z 293.864,A -85,B 0,C 180,E1 22400.047,E2 22400.047} C_VEL
LIN {X 0,Y 457.034,Z 293.862,A -85,B 0,C 180,E1 22396.332,E2 22396.332} C_VEL
LIN {X 0,Y 457.055,Z 293.861,A -85,B 0,C 180,E1 22392.691,E2 22392.691} C_VEL
LIN {X 0,Y 457.078,Z 293.86,A -85,B 0,C 180,E1 22388.976,E2 22388.976} C_VEL
LIN {X 0,Y 457.072,Z 293.866,A -85,B 0,C 180,E1 22385.302,E2 22385.302} C_VEL
LIN {X 0,Y 457.05,Z 293.864,A -85,B 0,C 180,E1 22381.658,E2 22381.658} C_VEL
LIN {X 0,Y 457.037,Z 293.863,A -85,B 0,C 180,E1 22378.033,E2 22378.033} C_VEL
LIN {X 0,Y 457.046,Z 293.861,A -85,B 0,C 180,E1 22374.414,E2 22374.414} C_VEL
LIN {X 0,Y 457.072,Z 293.859,A -85,B 0,C 180,E1 22370.745,E2 22370.745} C_VEL
LIN {X 0,Y 457.077,Z 293.863,A -85,B 0,C 180,E1 22367.119,E2 22367.119} C_VEL
LIN {X 0,Y 457.065,Z 293.866,A -85,B 0,C 180,E1 22363.381,E2 22363.381} C_VEL
LIN {X 0,Y 457.043,Z 293.866,A -85,B 0,C 180,E1 22359.836,E2 22359.836} C_VEL
LIN {X 0,Y 457.044,Z 293.866,A -85,B 0,C 180,E1 22356.171,E2 22356.171} C_VEL
LIN {X 0,Y 457.108,Z 294.088,A -85,B 0,C 180,E1 22353.095,E2 22353.095} C_VEL
LIN {X 0,Y 462.621,Z 314.397,A -85,B 0,C 180,E1 22349.805,E2 22349.805} C_VEL
LIN {X 0,Y 463.879,Z 320.513,A -85,B 0,C 180,E1 22348.867,E2 22348.867} C_VEL
LIN {X 0,Y 462.171,Z 348.756,A -85,B 0,C 180,E1 22345.086,E2 22345.086} C_VEL
LIN {X 0,Y 460.597,Z 378.252,A -85,B 0,C 180,E1 22341.198,E2 22341.198} C_VEL
LIN {X 0,Y 459.421,Z 403.622,A -85,B 0,C 180,E1 22337.931,E2 22337.931} C_VEL
LIN {X 0,Y 462.051,Z 421.956,A -85,B 0,C 180,E1 22337.452,E2 22337.452} C_VEL
LIN {X 0,Y 460.344,Z 523.504,A -85,B 0,C 180,E1 22335.533,E2 22335.533} C_VEL
LIN {X 0,Y 460.015,Z 538.78,A -85,B 0,C 180,E1 22335.02,E2 22335.02} C_VEL
LIN {X 0,Y 459.561,Z 553.947,A -85,B 0,C 180,E1 22334.268,E2 22334.268} C_VEL
LIN {X 0,Y 459.023,Z 568.434,A -85,B 0,C 180,E1 22333.283,E2 22333.283} C_VEL
LIN {X 0,Y 458.521,Z 580.666,A -85,B 0,C 180,E1 22332.209,E2 22332.209} C_VEL
LIN {X 0,Y 458.011,Z 592.63,A -85,B 0,C 180,E1 22330.883,E2 22330.883} C_VEL
LIN {X 0,Y 457.532,Z 603.723,A -85,B 0,C 180,E1 22329.304,E2 22329.304} C_VEL
LIN {X 0,Y 457.17,Z 612.6,A -85,B 0,C 180,E1 22327.665,E2 22327.665} C_VEL
LIN {X 0,Y 456.942,Z 619.412,A -85,B 0,C 180,E1 22326.027,E2 22326.027} C_VEL
LIN {X 0,Y 456.803,Z 624.784,A -85,B 0,C 180,E1 22324.266,E2 22324.266} C_VEL
LIN {X 0,Y 456.735,Z 628.306,A -85,B 0,C 180,E1 22322.508,E2 22322.508} C_VEL
LIN {X 0,Y 456.742,Z 630.285,A -85,B 0,C 180,E1 22320.625,E2 22320.625} C_VEL
LIN {X 0,Y 456.8,Z 630.365,A -85,B 0,C 180,E1 22318.744,E2 22318.744} C_VEL
LIN {X 0,Y 456.912,Z 628.761,A -85,B 0,C 180,E1 22316.988,E2 22316.988} C_VEL
LIN {X 0,Y 457.113,Z 625.167,A -85,B 0,C 180,E1 22315.105,E2 22315.105} C_VEL
LIN {X 0,Y 457.376,Z 619.861,A -85,B 0,C 180,E1 22313.345,E2 22313.345} C_VEL
LIN {X 0,Y 457.752,Z 613.009,A -85,B 0,C 180,E1 22311.686,E2 22311.686} C_VEL
LIN {X 0,Y 458.244,Z 604.197,A -85,B 0,C 180,E1 22310.073,E2 22310.073} C_VEL
LIN {X 0,Y 458.806,Z 593.988,A -85,B 0,C 180,E1 22308.624,E2 22308.624} C_VEL
LIN {X 0,Y 459.386,Z 582.799,A -85,B 0,C 180,E1 22307.363,E2 22307.363} C_VEL
LIN {X 0,Y 460.05,Z 569.193,A -85,B 0,C 180,E1 22306.167,E2 22306.167} C_VEL
LIN {X 0,Y 460.678,Z 554.147,A -85,B 0,C 180,E1 22305.159,E2 22305.159} C_VEL
LIN {X 0,Y 461.203,Z 538.644,A -85,B 0,C 180,E1 22304.404,E2 22304.404} C_VEL
LIN {X 0,Y 461.578,Z 523.073,A -85,B 0,C 180,E1 22303.889,E2 22303.889} C_VEL
LIN {X 0,Y 465.032,Z 429.052,A -85,B 0,C 180,E1 22301.655,E2 22301.655} C_VEL
LIN {X 0,Y 465.124,Z 421.573,A -85,B 0,C 180,E1 22301.456,E2 22301.456} C_VEL
LIN {X 0,Y 461.823,Z 403.434,A -85,B 0,C 180,E1 22300.684,E2 22300.684} C_VEL
LIN {X 0,Y 464.018,Z 375.235,A -85,B 0,C 180,E1 22296.775,E2 22296.775} C_VEL
LIN {X 0,Y 466.625,Z 348.903,A -85,B 0,C 180,E1 22292.981,E2 22292.981} C_VEL
LIN {X 0,Y 469.122,Z 329.559,A -85,B 0,C 180,E1 22290.083,E2 22290.083} C_VEL
LIN {X 0,Y 466.668,Z 319.358,A -85,B 0,C 180,E1 22287.902,E2 22287.902} C_VEL
LIN {X 0,Y 463.824,Z 310.529,A -85,B 0,C 180,E1 22285.611,E2 22285.611} C_VEL
LIN {X 0,Y 461.809,Z 305.184,A -85,B 0,C 180,E1 22283.919,E2 22283.919} C_VEL
LIN {X 0,Y 460.482,Z 301.815,A -85,B 0,C 180,E1 22282.629,E2 22282.629} C_VEL
LIN {X 0,Y 458.943,Z 298.093,A -85,B 0,C 180,E1 22280.816,E2 22280.816} C_VEL
LIN {X 0,Y 457.421,Z 295.4,A -85,B 0,C 180,E1 22278.355,E2 22278.355} C_VEL
LIN {X 0,Y 457.25,Z 294.826,A -85,B 0,C 180,E1 22276.369,E2 22276.369} C_VEL
LIN {X 0,Y 457.848,Z 296.433,A -85,B 0,C 180,E1 22274.159,E2 22274.159} C_VEL
LIN {X 0,Y 459.569,Z 299.129,A -85,B 0,C 180,E1 22272.291,E2 22272.291} C_VEL
LIN {X 0,Y 461.355,Z 302.906,A -85,B 0,C 180,E1 22270.719,E2 22270.719} C_VEL
LIN {X 0,Y 463.631,Z 308.492,A -85,B 0,C 180,E1 22269.031,E2 22269.031} C_VEL
LIN {X 0,Y 466.175,Z 314.574,A -85,B 0,C 180,E1 22267.527,E2 22267.527} C_VEL
LIN {X 0,Y 469.781,Z 324.809,A -85,B 0,C 180,E1 22265.525,E2 22265.525} C_VEL
LIN {X 0,Y 471.611,Z 331.827,A -85,B 0,C 180,E1 22264.404,E2 22264.404} C_VEL
LIN {X 0,Y 467.792,Z 361.667,A -85,B 0,C 180,E1 22261.364,E2 22261.364} C_VEL
LIN {X 0,Y 465.26,Z 390.491,A -85,B 0,C 180,E1 22258.66,E2 22258.66} C_VEL
LIN {X 0,Y 467.007,Z 407.902,A -85,B 0,C 180,E1 22258.193,E2 22258.193} C_VEL
LIN {X 0,Y 464.754,Z 529.917,A -85,B 0,C 180,E1 22256.023,E2 22256.023} C_VEL
LIN {X 0,Y 463.905,Z 589.912,A -85,B 0,C 180,E1 22255.01,E2 22255.01} C_VEL
LIN {X 0,Y 463.198,Z 609.065,A -85,B 0,C 180,E1 22254.46,E2 22254.46} C_VEL
LIN {X 0,Y 462.326,Z 627.756,A -85,B 0,C 180,E1 22253.686,E2 22253.686} C_VEL
LIN {X 0,Y 461.348,Z 645.843,A -85,B 0,C 180,E1 22252.693,E2 22252.693} C_VEL
LIN {X 0,Y 460.312,Z 663.388,A -85,B 0,C 180,E1 22251.47,E2 22251.47} C_VEL
LIN {X 0,Y 459.317,Z 679.866,A -85,B 0,C 180,E1 22250.052,E2 22250.052} C_VEL
LIN {X 0,Y 458.4,Z 695.459,A -85,B 0,C 180,E1 22248.409,E2 22248.409} C_VEL
LIN {X 0,Y 457.675,Z 708.52,A -85,B 0,C 180,E1 22246.762,E2 22246.762} C_VEL
LIN {X 0,Y 457.104,Z 720.502,A -85,B 0,C 180,E1 22244.959,E2 22244.959} C_VEL
LIN {X 0,Y 456.689,Z 731.211,A -85,B 0,C 180,E1 22243.024,E2 22243.024} C_VEL
LIN {X 0,Y 456.434,Z 740.443,A -85,B 0,C 180,E1 22240.988,E2 22240.988} C_VEL
LIN {X 0,Y 456.318,Z 748.262,A -85,B 0,C 180,E1 22238.824,E2 22238.824} C_VEL
LIN {X 0,Y 456.29,Z 754.218,A -85,B 0,C 180,E1 22236.67,E2 22236.67} C_VEL
LIN {X 0,Y 456.324,Z 758.551,A -85,B 0,C 180,E1 22234.464,E2 22234.464} C_VEL
LIN {X 0,Y 456.365,Z 761.175,A -85,B 0,C 180,E1 22232.261,E2 22232.261} C_VEL
LIN {X 0,Y 456.385,Z 762.135,A -85,B 0,C 180,E1 22230.001,E2 22230.001} C_VEL
LIN {X 0,Y 456.34,Z 761.354,A -85,B 0,C 180,E1 22227.741,E2 22227.741} C_VEL
LIN {X 0,Y 456.277,Z 758.832,A -85,B 0,C 180,E1 22225.476,E2 22225.476} C_VEL
LIN {X 0,Y 456.233,Z 754.519,A -85,B 0,C 180,E1 22223.204,E2 22223.204} C_VEL
LIN {X 0,Y 456.269,Z 748.295,A -85,B 0,C 180,E1 22220.923,E2 22220.923} C_VEL
LIN {X 0,Y 456.404,Z 740.509,A -85,B 0,C 180,E1 22218.758,E2 22218.758} C_VEL
LIN {X 0,Y 456.709,Z 731.289,A -85,B 0,C 180,E1 22216.711,E2 22216.711} C_VEL
LIN {X 0,Y 457.182,Z 720.711,A -85,B 0,C 180,E1 22214.786,E2 22214.786} C_VEL
LIN {X 0,Y 457.893,Z 707.851,A -85,B 0,C 180,E1 22212.856,E2 22212.856} C_VEL
LIN {X 0,Y 458.732,Z 694.404,A -85,B 0,C 180,E1 22211.182,E2 22211.182} C_VEL
LIN {X 0,Y 459.703,Z 679.371,A -85,B 0,C 180,E1 22209.626,E2 22209.626} C_VEL
LIN {X 0,Y 460.785,Z 662.817,A -85,B 0,C 180,E1 22208.221,E2 22208.221} C_VEL
LIN {X 0,Y 461.83,Z 645.991,A -85,B 0,C 180,E1 22207.065,E2 22207.065} C_VEL
LIN {X 0,Y 462.829,Z 628.294,A -85,B 0,C 180,E1 22206.106,E2 22206.106} C_VEL
LIN {X 0,Y 463.701,Z 609.93,A -85,B 0,C 180,E1 22205.358,E2 22205.358} C_VEL
LIN {X 0,Y 464.387,Z 591.001,A -85,B 0,C 180,E1 22204.827,E2 22204.827} C_VEL
LIN {X 0,Y 466.962,Z 404.941,A -85,B 0,C 180,E1 22201.713,E2 22201.713} C_VEL
LIN {X 0,Y 464.884,Z 387.449,A -85,B 0,C 180,E1 22201.27,E2 22201.27} C_VEL
LIN {X 0,Y 467.987,Z 342.416,A -85,B 0,C 180,E1 22197.281,E2 22197.281} C_VEL
LIN {X 0,Y 468.895,Z 327.669,A -85,B 0,C 180,E1 22195.939,E2 22195.939} C_VEL
LIN {X 0,Y 460.204,Z 302.985,A -85,B 0,C 180,E1 22192.845,E2 22192.845} C_VEL
LIN {X 0,Y 457.048,Z 293.868,A -85,B 0,C 180,E1 22191.631,E2 22191.631} C_VEL
LIN {X 0,Y 457.038,Z 293.869,A -85,B 0,C 180,E1 22187.978,E2 22187.978} C_VEL
LIN {X 0,Y 457.003,Z 293.871,A -85,B 0,C 180,E1 22184.437,E2 22184.437} C_VEL
LIN {X 0,Y 456.996,Z 293.87,A -85,B 0,C 180,E1 22180.8,E2 22180.8} C_VEL
LIN {X 0,Y 457.013,Z 293.867,A -85,B 0,C 180,E1 22177.218,E2 22177.218} C_VEL
LIN {X 0,Y 457.048,Z 293.867,A -85,B 0,C 180,E1 22173.607,E2 22173.607} C_VEL
LIN {X 0,Y 457.042,Z 293.867,A -85,B 0,C 180,E1 22169.921,E2 22169.921} C_VEL
LIN {X 0,Y 457.008,Z 293.867,A -85,B 0,C 180,E1 22166.369,E2 22166.369} C_VEL
LIN {X 0,Y 457.004,Z 293.866,A -85,B 0,C 180,E1 22162.785,E2 22162.785} C_VEL
LIN {X 0,Y 457.032,Z 293.866,A -85,B 0,C 180,E1 22159.291,E2 22159.291} C_VEL
LIN {X 0,Y 457.063,Z 293.866,A -85,B 0,C 180,E1 22155.611,E2 22155.611} C_VEL
LIN {X 0,Y 457.03,Z 293.867,A -85,B 0,C 180,E1 22151.997,E2 22151.997} C_VEL
LIN {X 0,Y 457.006,Z 293.866,A -85,B 0,C 180,E1 22148.431,E2 22148.431} C_VEL
LIN {X 0,Y 457.008,Z 293.866,A -85,B 0,C 180,E1 22144.771,E2 22144.771} C_VEL
LIN {X 0,Y 457.04,Z 293.865,A -85,B 0,C 180,E1 22141.255,E2 22141.255} C_VEL
LIN {X 0,Y 457.06,Z 293.868,A -85,B 0,C 180,E1 22137.62,E2 22137.62} C_VEL
LIN {X 0,Y 457.032,Z 293.866,A -85,B 0,C 180,E1 22133.974,E2 22133.974} C_VEL
LIN {X 0,Y 457.01,Z 293.866,A -85,B 0,C 180,E1 22130.431,E2 22130.431} C_VEL
LIN {X 0,Y 457.015,Z 293.865,A -85,B 0,C 180,E1 22126.722,E2 22126.722} C_VEL
LIN {X 0,Y 457.048,Z 293.864,A -85,B 0,C 180,E1 22123.218,E2 22123.218} C_VEL
LIN {X 0,Y 457.068,Z 293.866,A -85,B 0,C 180,E1 22119.515,E2 22119.515} C_VEL
LIN {X 0,Y 457.03,Z 293.866,A -85,B 0,C 180,E1 22115.991,E2 22115.991} C_VEL
LIN {X 0,Y 457.016,Z 293.865,A -85,B 0,C 180,E1 22112.369,E2 22112.369} C_VEL
LIN {X 0,Y 457.019,Z 293.864,A -85,B 0,C 180,E1 22108.624,E2 22108.624} C_VEL
LIN {X 0,Y 457.042,Z 293.863,A -85,B 0,C 180,E1 22105.031,E2 22105.031} C_VEL
LIN {X 0,Y 457.075,Z 293.863,A -85,B 0,C 180,E1 22101.345,E2 22101.345} C_VEL
LIN {X 0,Y 457.043,Z 293.866,A -85,B 0,C 180,E1 22097.812,E2 22097.812} C_VEL
LIN {X 0,Y 457.021,Z 293.865,A -85,B 0,C 180,E1 22094.257,E2 22094.257} C_VEL
LIN {X 0,Y 457.022,Z 293.864,A -85,B 0,C 180,E1 22090.523,E2 22090.523} C_VEL
LIN {X 0,Y 457.048,Z 293.863,A -85,B 0,C 180,E1 22086.983,E2 22086.983} C_VEL
LIN {X 0,Y 457.072,Z 293.863,A -85,B 0,C 180,E1 22083.302,E2 22083.302} C_VEL
LIN {X 0,Y 457.056,Z 293.866,A -85,B 0,C 180,E1 22079.629,E2 22079.629} C_VEL
LIN {X 0,Y 457.028,Z 293.865,A -85,B 0,C 180,E1 22076.086,E2 22076.086} C_VEL
LIN {X 0,Y 457.026,Z 293.863,A -85,B 0,C 180,E1 22072.374,E2 22072.374} C_VEL
LIN {X 0,Y 457.042,Z 293.862,A -85,B 0,C 180,E1 22068.758,E2 22068.758} C_VEL
LIN {X 0,Y 457.077,Z 293.864,A -85,B 0,C 180,E1 22065.334,E2 22065.334} C_VEL
LIN {X 0,Y 456.126,Z 293.976,A -85,B 0,C 180,E1 22064.369,E2 22064.369} C_VEL
LIN {X 0,Y 449.596,Z 294.797,A -85,B 0,C 180,E1 22061.582,E2 22061.582} C_VEL
LIN {X 0,Y 449.119,Z 294.851,A -85,B 0,C 180,E1 22060.943,E2 22060.943} C_VEL
LIN {X 0,Y 449.141,Z 294.85,A -85,B 0,C 180,E1 22057.16,E2 22057.16} C_VEL
LIN {X 0,Y 449.125,Z 294.856,A -85,B 0,C 180,E1 22053.445,E2 22053.445} C_VEL
LIN {X 0,Y 449.099,Z 294.853,A -85,B 0,C 180,E1 22049.871,E2 22049.871} C_VEL
LIN {X 0,Y 449.092,Z 294.852,A -85,B 0,C 180,E1 22046.169,E2 22046.169} C_VEL
LIN {X 0,Y 449.098,Z 294.851,A -85,B 0,C 180,E1 22042.451,E2 22042.451} C_VEL
LIN {X 0,Y 449.121,Z 294.85,A -85,B 0,C 180,E1 22038.831,E2 22038.831} C_VEL
LIN {X 0,Y 449.144,Z 294.851,A -85,B 0,C 180,E1 22035.166,E2 22035.166} C_VEL
LIN {X 0,Y 449.125,Z 294.855,A -85,B 0,C 180,E1 22031.436,E2 22031.436} C_VEL
LIN {X 0,Y 449.104,Z 294.853,A -85,B 0,C 180,E1 22027.76,E2 22027.76} C_VEL
LIN {X 0,Y 449.097,Z 294.852,A -85,B 0,C 180,E1 22024.08,E2 22024.08} C_VEL
LIN {X 0,Y 449.104,Z 294.85,A -85,B 0,C 180,E1 22020.379,E2 22020.379} C_VEL
LIN {X 0,Y 449.129,Z 294.849,A -85,B 0,C 180,E1 22016.793,E2 22016.793} C_VEL
LIN {X 0,Y 449.139,Z 294.851,A -85,B 0,C 180,E1 22013.048,E2 22013.048} C_VEL
LIN {X 0,Y 449.135,Z 294.855,A -85,B 0,C 180,E1 22009.286,E2 22009.286} C_VEL
LIN {X 0,Y 449.113,Z 294.853,A -85,B 0,C 180,E1 22005.61,E2 22005.61} C_VEL
LIN {X 0,Y 449.102,Z 294.852,A -85,B 0,C 180,E1 22001.902,E2 22001.902} C_VEL
LIN {X 0,Y 449.105,Z 294.854,A -85,B 0,C 180,E1 21998.195,E2 21998.195} C_VEL
LIN {X 0,Y 449.123,Z 294.853,A -85,B 0,C 180,E1 21994.541,E2 21994.541} C_VEL
LIN {X 0,Y 449.127,Z 294.956,A -85,B 0,C 180,E1 21993.574,E2 21993.574} C_VEL
LIN {X 0,Y 454.693,Z 315.359,A -85,B 0,C 180,E1 21990.208,E2 21990.208} C_VEL
LIN {X 0,Y 456.294,Z 322.858,A -85,B 0,C 180,E1 21989.035,E2 21989.035} C_VEL
LIN {X 0,Y 454.483,Z 351.199,A -85,B 0,C 180,E1 21985.192,E2 21985.192} C_VEL
LIN {X 0,Y 452.832,Z 380.474,A -85,B 0,C 180,E1 21981.284,E2 21981.284} C_VEL
LIN {X 0,Y 451.698,Z 403.555,A -85,B 0,C 180,E1 21978.276,E2 21978.276} C_VEL
LIN {X 0,Y 454.458,Z 422.906,A -85,B 0,C 180,E1 21977.757,E2 21977.757} C_VEL
LIN {X 0,Y 452.619,Z 524.194,A -85,B 0,C 180,E1 21975.785,E2 21975.785} C_VEL
LIN {X 0,Y 452.266,Z 539.657,A -85,B 0,C 180,E1 21975.251,E2 21975.251} C_VEL
LIN {X 0,Y 451.788,Z 554.864,A -85,B 0,C 180,E1 21974.48,E2 21974.48} C_VEL
LIN {X 0,Y 451.211,Z 569.681,A -85,B 0,C 180,E1 21973.452,E2 21973.452} C_VEL
LIN {X 0,Y 450.658,Z 582.461,A -85,B 0,C 180,E1 21972.296,E2 21972.296} C_VEL
LIN {X 0,Y 450.15,Z 593.768,A -85,B 0,C 180,E1 21971.01,E2 21971.01} C_VEL
LIN {X 0,Y 449.666,Z 604.479,A -85,B 0,C 180,E1 21969.469,E2 21969.469} C_VEL
LIN {X 0,Y 449.282,Z 613.462,A -85,B 0,C 180,E1 21967.8,E2 21967.8} C_VEL
LIN {X 0,Y 449.039,Z 620.361,A -85,B 0,C 180,E1 21966.134,E2 21966.134} C_VEL
LIN {X 0,Y 448.889,Z 625.814,A -85,B 0,C 180,E1 21964.341,E2 21964.341} C_VEL
LIN {X 0,Y 448.818,Z 629.411,A -85,B 0,C 180,E1 21962.552,E2 21962.552} C_VEL
LIN {X 0,Y 448.829,Z 631.458,A -85,B 0,C 180,E1 21960.636,E2 21960.636} C_VEL
LIN {X 0,Y 448.896,Z 631.589,A -85,B 0,C 180,E1 21958.722,E2 21958.722} C_VEL
LIN {X 0,Y 449.025,Z 630.036,A -85,B 0,C 180,E1 21956.935,E2 21956.935} C_VEL
LIN {X 0,Y 449.252,Z 626.492,A -85,B 0,C 180,E1 21955.019,E2 21955.019} C_VEL
LIN {X 0,Y 449.551,Z 621.251,A -85,B 0,C 180,E1 21953.229,E2 21953.229} C_VEL
LIN {X 0,Y 449.959,Z 614.551,A -85,B 0,C 180,E1 21951.565,E2 21951.565} C_VEL
LIN {X 0,Y 450.495,Z 605.645,A -85,B 0,C 180,E1 21949.9,E2 21949.9} C_VEL
LIN {X 0,Y 451.1,Z 595.568,A -85,B 0,C 180,E1 21948.436,E2 21948.436} C_VEL
LIN {X 0,Y 451.739,Z 584.471,A -85,B 0,C 180,E1 21947.146,E2 21947.146} C_VEL
LIN {X 0,Y 452.452,Z 571.077,A -85,B 0,C 180,E1 21945.93,E2 21945.93} C_VEL
LIN {X 0,Y 453.08,Z 557.37,A -85,B 0,C 180,E1 21944.97,E2 21944.97} C_VEL
LIN {X 0,Y 453.622,Z 543.284,A -85,B 0,C 180,E1 21944.219,E2 21944.219} C_VEL
LIN {X 0,Y 454.112,Z 526.353,A -85,B 0,C 180,E1 21943.592,E2 21943.592} C_VEL
LIN {X 0,Y 457.999,Z 429.837,A -85,B 0,C 180,E1 21941.189,E2 21941.189} C_VEL
LIN {X 0,Y 458.108,Z 422.919,A -85,B 0,C 180,E1 21940.993,E2 21940.993} C_VEL
LIN {X 0,Y 454.551,Z 403.47,A -85,B 0,C 180,E1 21940.131,E2 21940.131} C_VEL
LIN {X 0,Y 457.036,Z 375.213,A -85,B 0,C 180,E1 21936.125,E2 21936.125} C_VEL
LIN {X 0,Y 460.007,Z 348.76,A -85,B 0,C 180,E1 21932.209,E2 21932.209} C_VEL
LIN {X 0,Y 462.176,Z 332.531,A -85,B 0,C 180,E1 21929.677,E2 21929.677} C_VEL
LIN {X 0,Y 459.918,Z 322.933,A -85,B 0,C 180,E1 21927.514,E2 21927.514} C_VEL
LIN {X 0,Y 457.214,Z 314.114,A -85,B 0,C 180,E1 21925.093,E2 21925.093} C_VEL
LIN {X 0,Y 454.976,Z 307.74,A -85,B 0,C 180,E1 21922.817,E2 21922.817} C_VEL
LIN {X 0,Y 453.216,Z 303.661,A -85,B 0,C 180,E1 21920.715,E2 21920.715} C_VEL
LIN {X 0,Y 451.907,Z 301.062,A -85,B 0,C 180,E1 21918.072,E2 21918.072} C_VEL
LIN {X 0,Y 451.889,Z 300.811,A -85,B 0,C 180,E1 21916.164,E2 21916.164} C_VEL
LIN {X 0,Y 452.513,Z 302.451,A -85,B 0,C 180,E1 21914.1,E2 21914.1} C_VEL
LIN {X 0,Y 454.045,Z 304.94,A -85,B 0,C 180,E1 21912.366,E2 21912.366} C_VEL
LIN {X 0,Y 456.053,Z 309.638,A -85,B 0,C 180,E1 21910.464,E2 21910.464} C_VEL
LIN {X 0,Y 458.136,Z 314.674,A -85,B 0,C 180,E1 21908.944,E2 21908.944} C_VEL
LIN {X 0,Y 461.033,Z 322.071,A -85,B 0,C 180,E1 21907.153,E2 21907.153} C_VEL
LIN {X 0,Y 464.155,Z 332.059,A -85,B 0,C 180,E1 21905.263,E2 21905.263} C_VEL
LIN {X 0,Y 464.802,Z 335.394,A -85,B 0,C 180,E1 21904.739,E2 21904.739} C_VEL
LIN {X 0,Y 460.681,Z 364.53,A -85,B 0,C 180,E1 21901.685,E2 21901.685} C_VEL
LIN {X 0,Y 458.124,Z 390.81,A -85,B 0,C 180,E1 21899.149,E2 21899.149} C_VEL
LIN {X 0,Y 459.908,Z 408.819,A -85,B 0,C 180,E1 21898.639,E2 21898.639} C_VEL
LIN {X 0,Y 457.423,Z 527.22,A -85,B 0,C 180,E1 21896.457,E2 21896.457} C_VEL
LIN {X 0,Y 456.441,Z 589.137,A -85,B 0,C 180,E1 21895.379,E2 21895.379} C_VEL
LIN {X 0,Y 455.681,Z 608.201,A -85,B 0,C 180,E1 21894.822,E2 21894.822} C_VEL
LIN {X 0,Y 454.701,Z 627.471,A -85,B 0,C 180,E1 21894.005,E2 21894.005} C_VEL
LIN {X 0,Y 453.689,Z 644.838,A -85,B 0,C 180,E1 21893.029,E2 21893.029} C_VEL
LIN {X 0,Y 452.586,Z 662.351,A -85,B 0,C 180,E1 21891.787,E2 21891.787} C_VEL
LIN {X 0,Y 451.516,Z 678.805,A -85,B 0,C 180,E1 21890.346,E2 21890.346} C_VEL
LIN {X 0,Y 450.552,Z 694.139,A -85,B 0,C 180,E1 21888.704,E2 21888.704} C_VEL
LIN {X 0,Y 449.735,Z 707.894,A -85,B 0,C 180,E1 21886.933,E2 21886.933} C_VEL
LIN {X 0,Y 449.103,Z 720.559,A -85,B 0,C 180,E1 21884.968,E2 21884.968} C_VEL
LIN {X 0,Y 448.672,Z 731.645,A -85,B 0,C 180,E1 21882.877,E2 21882.877} C_VEL
LIN {X 0,Y 448.428,Z 741.125,A -85,B 0,C 180,E1 21880.666,E2 21880.666} C_VEL
LIN {X 0,Y 448.346,Z 748.55,A -85,B 0,C 180,E1 21878.465,E2 21878.465} C_VEL
LIN {X 0,Y 448.348,Z 754.135,A -85,B 0,C 180,E1 21876.274,E2 21876.274} C_VEL
LIN {X 0,Y 448.405,Z 758.015,A -85,B 0,C 180,E1 21874.093,E2 21874.093} C_VEL
LIN {X 0,Y 448.454,Z 760.361,A -85,B 0,C 180,E1 21871.79,E2 21871.79} C_VEL
LIN {X 0,Y 448.453,Z 760.949,A -85,B 0,C 180,E1 21869.49,E2 21869.49} C_VEL
LIN {X 0,Y 448.402,Z 759.787,A -85,B 0,C 180,E1 21867.189,E2 21867.189} C_VEL
LIN {X 0,Y 448.329,Z 756.862,A -85,B 0,C 180,E1 21864.883,E2 21864.883} C_VEL
LIN {X 0,Y 448.276,Z 752.108,A -85,B 0,C 180,E1 21862.568,E2 21862.568} C_VEL
LIN {X 0,Y 448.318,Z 745.406,A -85,B 0,C 180,E1 21860.242,E2 21860.242} C_VEL
LIN {X 0,Y 448.501,Z 737.113,A -85,B 0,C 180,E1 21858.035,E2 21858.035} C_VEL
LIN {X 0,Y 448.877,Z 727.313,A -85,B 0,C 180,E1 21855.95,E2 21855.95} C_VEL
LIN {X 0,Y 449.445,Z 715.891,A -85,B 0,C 180,E1 21853.958,E2 21853.958} C_VEL
LIN {X 0,Y 450.207,Z 703.413,A -85,B 0,C 180,E1 21852.154,E2 21852.154} C_VEL
LIN {X 0,Y 451.15,Z 689.271,A -85,B 0,C 180,E1 21850.45,E2 21850.45} C_VEL
LIN {X 0,Y 452.242,Z 673.429,A -85,B 0,C 180,E1 21848.878,E2 21848.878} C_VEL
LIN {X 0,Y 453.397,Z 656.529,A -85,B 0,C 180,E1 21847.52,E2 21847.52} C_VEL
LIN {X 0,Y 454.504,Z 639.103,A -85,B 0,C 180,E1 21846.399,E2 21846.399} C_VEL
LIN {X 0,Y 455.52,Z 620.888,A -85,B 0,C 180,E1 21845.491,E2 21845.491} C_VEL
LIN {X 0,Y 456.388,Z 601.851,A -85,B 0,C 180,E1 21844.801,E2 21844.801} C_VEL
LIN {X 0,Y 456.977,Z 582.755,A -85,B 0,C 180,E1 21844.352,E2 21844.352} C_VEL
LIN {X 0,Y 459.665,Z 406.647,A -85,B 0,C 180,E1 21841.366,E2 21841.366} C_VEL
LIN {X 0,Y 457.423,Z 387.685,A -85,B 0,C 180,E1 21840.882,E2 21840.882} C_VEL
LIN {X 0,Y 460.703,Z 342.852,A -85,B 0,C 180,E1 21836.846,E2 21836.846} C_VEL
LIN {X 0,Y 461.684,Z 330.783,A -85,B 0,C 180,E1 21835.733,E2 21835.733} C_VEL
LIN {X 0,Y 453.469,Z 307.344,A -85,B 0,C 180,E1 21832.748,E2 21832.748} C_VEL
LIN {X 0,Y 449.066,Z 294.86,A -85,B 0,C 180,E1 21831.067,E2 21831.067} C_VEL
LIN {X 0,Y 449.093,Z 294.858,A -85,B 0,C 180,E1 21827.472,E2 21827.472} C_VEL
LIN {X 0,Y 449.109,Z 294.858,A -85,B 0,C 180,E1 21823.82,E2 21823.82} C_VEL
LIN {X 0,Y 449.077,Z 294.859,A -85,B 0,C 180,E1 21820.212,E2 21820.212} C_VEL
LIN {X 0,Y 449.058,Z 294.856,A -85,B 0,C 180,E1 21816.637,E2 21816.637} C_VEL
LIN {X 0,Y 449.064,Z 294.856,A -85,B 0,C 180,E1 21812.908,E2 21812.908} C_VEL
LIN {X 0,Y 449.091,Z 294.855,A -85,B 0,C 180,E1 21809.329,E2 21809.329} C_VEL
LIN {X 0,Y 449.115,Z 294.856,A -85,B 0,C 180,E1 21805.628,E2 21805.628} C_VEL
LIN {X 0,Y 449.095,Z 294.856,A -85,B 0,C 180,E1 21801.966,E2 21801.966} C_VEL
LIN {X 0,Y 449.068,Z 294.855,A -85,B 0,C 180,E1 21798.433,E2 21798.433} C_VEL
LIN {X 0,Y 449.064,Z 294.855,A -85,B 0,C 180,E1 21794.706,E2 21794.706} C_VEL
LIN {X 0,Y 449.086,Z 294.855,A -85,B 0,C 180,E1 21791.17,E2 21791.17} C_VEL
LIN {X 0,Y 449.13,Z 294.854,A -85,B 0,C 180,E1 21787.549,E2 21787.549} C_VEL
LIN {X 0,Y 449.105,Z 294.856,A -85,B 0,C 180,E1 21783.831,E2 21783.831} C_VEL
LIN {X 0,Y 449.075,Z 294.855,A -85,B 0,C 180,E1 21780.257,E2 21780.257} C_VEL
LIN {X 0,Y 449.07,Z 294.855,A -85,B 0,C 180,E1 21776.555,E2 21776.555} C_VEL
LIN {X 0,Y 449.077,Z 294.854,A -85,B 0,C 180,E1 21772.84,E2 21772.84} C_VEL
LIN {X 0,Y 449.104,Z 294.854,A -85,B 0,C 180,E1 21769.224,E2 21769.224} C_VEL
LIN {X 0,Y 449.133,Z 294.854,A -85,B 0,C 180,E1 21765.552,E2 21765.552} C_VEL
LIN {X 0,Y 449.102,Z 294.855,A -85,B 0,C 180,E1 21761.841,E2 21761.841} C_VEL
LIN {X 0,Y 449.077,Z 294.854,A -85,B 0,C 180,E1 21758.312,E2 21758.312} C_VEL
LIN {X 0,Y 449.076,Z 294.854,A -85,B 0,C 180,E1 21754.553,E2 21754.553} C_VEL
LIN {X 0,Y 449.095,Z 294.853,A -85,B 0,C 180,E1 21750.967,E2 21750.967} C_VEL
LIN {X 0,Y 449.131,Z 294.853,A -85,B 0,C 180,E1 21747.405,E2 21747.405} C_VEL
LIN {X 0,Y 449.113,Z 294.855,A -85,B 0,C 180,E1 21743.69,E2 21743.69} C_VEL
LIN {X 0,Y 449.083,Z 294.854,A -85,B 0,C 180,E1 21740.121,E2 21740.121} C_VEL
LIN {X 0,Y 449.081,Z 294.853,A -85,B 0,C 180,E1 21736.534,E2 21736.534} C_VEL
LIN {X 0,Y 449.101,Z 294.852,A -85,B 0,C 180,E1 21732.91,E2 21732.91} C_VEL
LIN {X 0,Y 449.131,Z 294.851,A -85,B 0,C 180,E1 21729.225,E2 21729.225} C_VEL
LIN {X 0,Y 449.128,Z 294.855,A -85,B 0,C 180,E1 21725.438,E2 21725.438} C_VEL
LIN {X 0,Y 449.109,Z 294.854,A -85,B 0,C 180,E1 21721.745,E2 21721.745} C_VEL
LIN {X 0,Y 449.087,Z 294.853,A -85,B 0,C 180,E1 21718.163,E2 21718.163} C_VEL
LIN {X 0,Y 449.087,Z 294.852,A -85,B 0,C 180,E1 21714.418,E2 21714.418} C_VEL
LIN {X 0,Y 449.104,Z 294.851,A -85,B 0,C 180,E1 21710.77,E2 21710.77} C_VEL
LIN {X 0,Y 449.128,Z 294.851,A -85,B 0,C 180,E1 21707.088,E2 21707.088} C_VEL
LIN {X 0,Y 449.135,Z 294.854,A -85,B 0,C 180,E1 21703.386,E2 21703.386} C_VEL
LIN {X 0,Y 449.119,Z 294.851,A -85,B 0,C 180,E1 21700.943,E2 21700.943} C_VEL
LIN {X 0,Y 448.089,Z 294.98,A -85,B 0,C 180,E1 21699.961,E2 21699.961} C_VEL
LIN {X 0,Y 441.601,Z 295.789,A -85,B 0,C 180,E1 21697.123,E2 21697.123} C_VEL
LIN {X 0,Y 441.155,Z 295.841,A -85,B 0,C 180,E1 21696.473,E2 21696.473} C_VEL
LIN {X 0,Y 441.177,Z 295.84,A -85,B 0,C 180,E1 21692.857,E2 21692.857} C_VEL
LIN {X 0,Y 441.196,Z 295.839,A -85,B 0,C 180,E1 21689.09,E2 21689.09} C_VEL
LIN {X 0,Y 441.191,Z 295.843,A -85,B 0,C 180,E1 21685.319,E2 21685.319} C_VEL
LIN {X 0,Y 441.171,Z 295.843,A -85,B 0,C 180,E1 21681.659,E2 21681.659} C_VEL
LIN {X 0,Y 441.157,Z 295.842,A -85,B 0,C 180,E1 21677.964,E2 21677.964} C_VEL
LIN {X 0,Y 441.156,Z 295.841,A -85,B 0,C 180,E1 21674.217,E2 21674.217} C_VEL
LIN {X 0,Y 441.169,Z 295.839,A -85,B 0,C 180,E1 21670.521,E2 21670.521} C_VEL
LIN {X 0,Y 441.197,Z 295.838,A -85,B 0,C 180,E1 21666.916,E2 21666.916} C_VEL
LIN {X 0,Y 441.198,Z 295.841,A -85,B 0,C 180,E1 21663.192,E2 21663.192} C_VEL
LIN {X 0,Y 441.186,Z 295.843,A -85,B 0,C 180,E1 21659.445,E2 21659.445} C_VEL
LIN {X 0,Y 441.165,Z 295.842,A -85,B 0,C 180,E1 21655.8,E2 21655.8} C_VEL
LIN {X 0,Y 441.162,Z 295.84,A -85,B 0,C 180,E1 21652.061,E2 21652.061} C_VEL
LIN {X 0,Y 441.171,Z 295.839,A -85,B 0,C 180,E1 21648.39,E2 21648.39} C_VEL
LIN {X 0,Y 441.187,Z 295.84,A -85,B 0,C 180,E1 21644.628,E2 21644.628} C_VEL
LIN {X 0,Y 441.203,Z 295.839,A -85,B 0,C 180,E1 21640.806,E2 21640.806} C_VEL
LIN {X 0,Y 441.197,Z 295.841,A -85,B 0,C 180,E1 21637.069,E2 21637.069} C_VEL
LIN {X 0,Y 441.188,Z 296.003,A -85,B 0,C 180,E1 21634.037,E2 21634.037} C_VEL
LIN {X 0,Y 446.642,Z 315.914,A -85,B 0,C 180,E1 21630.688,E2 21630.688} C_VEL
LIN {X 0,Y 448.745,Z 324.702,A -85,B 0,C 180,E1 21629.277,E2 21629.277} C_VEL
LIN {X 0,Y 446.819,Z 353.106,A -85,B 0,C 180,E1 21625.371,E2 21625.371} C_VEL
LIN {X 0,Y 445.105,Z 381.908,A -85,B 0,C 180,E1 21621.476,E2 21621.476} C_VEL
LIN {X 0,Y 443.982,Z 403.443,A -85,B 0,C 180,E1 21618.631,E2 21618.631} C_VEL
LIN {X 0,Y 446.872,Z 423.815,A -85,B 0,C 180,E1 21618.071,E2 21618.071} C_VEL
LIN {X 0,Y 444.906,Z 524.703,A -85,B 0,C 180,E1 21616.049,E2 21616.049} C_VEL
LIN {X 0,Y 444.547,Z 539.805,A -85,B 0,C 180,E1 21615.522,E2 21615.522} C_VEL
LIN {X 0,Y 444.043,Z 555.135,A -85,B 0,C 180,E1 21614.738,E2 21614.738} C_VEL
LIN {X 0,Y 443.437,Z 570.088,A -85,B 0,C 180,E1 21613.693,E2 21613.693} C_VEL
LIN {X 0,Y 442.854,Z 583.004,A -85,B 0,C 180,E1 21612.516,E2 21612.516} C_VEL
LIN {X 0,Y 442.295,Z 594.837,A -85,B 0,C 180,E1 21611.152,E2 21611.152} C_VEL
LIN {X 0,Y 441.804,Z 605.23,A -85,B 0,C 180,E1 21609.639,E2 21609.639} C_VEL
LIN {X 0,Y 441.398,Z 614.324,A -85,B 0,C 180,E1 21607.94,E2 21607.94} C_VEL
LIN {X 0,Y 441.138,Z 621.315,A -85,B 0,C 180,E1 21606.244,E2 21606.244} C_VEL
LIN {X 0,Y 440.97,Z 627.171,A -85,B 0,C 180,E1 21604.289,E2 21604.289} C_VEL
LIN {X 0,Y 440.9,Z 630.907,A -85,B 0,C 180,E1 21602.338,E2 21602.338} C_VEL
LIN {X 0,Y 440.919,Z 632.691,A -85,B 0,C 180,E1 21600.518,E2 21600.518} C_VEL
LIN {X 0,Y 441.005,Z 632.795,A -85,B 0,C 180,E1 21598.569,E2 21598.569} C_VEL
LIN {X 0,Y 441.155,Z 631.158,A -85,B 0,C 180,E1 21596.75,E2 21596.75} C_VEL
LIN {X 0,Y 441.396,Z 627.839,A -85,B 0,C 180,E1 21594.93,E2 21594.93} C_VEL
LIN {X 0,Y 441.728,Z 622.639,A -85,B 0,C 180,E1 21593.108,E2 21593.108} C_VEL
LIN {X 0,Y 442.178,Z 615.996,A -85,B 0,C 180,E1 21591.415,E2 21591.415} C_VEL
LIN {X 0,Y 442.768,Z 607.184,A -85,B 0,C 180,E1 21589.722,E2 21589.722} C_VEL
LIN {X 0,Y 443.432,Z 597.162,A -85,B 0,C 180,E1 21588.224,E2 21588.224} C_VEL
LIN {X 0,Y 444.148,Z 585.601,A -85,B 0,C 180,E1 21586.856,E2 21586.856} C_VEL
LIN {X 0,Y 444.931,Z 571.915,A -85,B 0,C 180,E1 21585.596,E2 21585.596} C_VEL
LIN {X 0,Y 445.646,Z 557.609,A -85,B 0,C 180,E1 21584.58,E2 21584.58} C_VEL
LIN {X 0,Y 446.271,Z 542.474,A -85,B 0,C 180,E1 21583.777,E2 21583.777} C_VEL
LIN {X 0,Y 446.77,Z 526.672,A -85,B 0,C 180,E1 21583.189,E2 21583.189} C_VEL
LIN {X 0,Y 451.019,Z 431.611,A -85,B 0,C 180,E1 21580.719,E2 21580.719} C_VEL
LIN {X 0,Y 451.176,Z 424.303,A -85,B 0,C 180,E1 21580.509,E2 21580.509} C_VEL
LIN {X 0,Y 447.366,Z 403.339,A -85,B 0,C 180,E1 21579.516,E2 21579.516} C_VEL
LIN {X 0,Y 450.016,Z 376.248,A -85,B 0,C 180,E1 21575.589,E2 21575.589} C_VEL
LIN {X 0,Y 453.286,Z 350.359,A -85,B 0,C 180,E1 21571.658,E2 21571.658} C_VEL
LIN {X 0,Y 455.408,Z 336.166,A -85,B 0,C 180,E1 21569.377,E2 21569.377} C_VEL
LIN {X 0,Y 453.28,Z 326.671,A -85,B 0,C 180,E1 21567.136,E2 21567.136} C_VEL
LIN {X 0,Y 450.995,Z 318.972,A -85,B 0,C 180,E1 21564.894,E2 21564.894} C_VEL
LIN {X 0,Y 448.985,Z 312.987,A -85,B 0,C 180,E1 21562.658,E2 21562.658} C_VEL
LIN {X 0,Y 447.531,Z 309.268,A -85,B 0,C 180,E1 21560.616,E2 21560.616} C_VEL
LIN {X 0,Y 446.446,Z 306.949,A -85,B 0,C 180,E1 21558.132,E2 21558.132} C_VEL
LIN {X 0,Y 446.478,Z 306.713,A -85,B 0,C 180,E1 21556.146,E2 21556.146} C_VEL
LIN {X 0,Y 447.212,Z 308.554,A -85,B 0,C 180,E1 21553.951,E2 21553.951} C_VEL
LIN {X 0,Y 448.505,Z 310.727,A -85,B 0,C 180,E1 21552.446,E2 21552.446} C_VEL
LIN {X 0,Y 450.358,Z 315.174,A -85,B 0,C 180,E1 21550.597,E2 21550.597} C_VEL
LIN {X 0,Y 452.788,Z 321.032,A -85,B 0,C 180,E1 21548.784,E2 21548.784} C_VEL
LIN {X 0,Y 455.726,Z 329.616,A -85,B 0,C 180,E1 21546.792,E2 21546.792} C_VEL
LIN {X 0,Y 458.19,Z 338.259,A -85,B 0,C 180,E1 21545.178,E2 21545.178} C_VEL
LIN {X 0,Y 453.807,Z 366.312,A -85,B 0,C 180,E1 21542.148,E2 21542.148} C_VEL
LIN {X 0,Y 451.083,Z 391.199,A -85,B 0,C 180,E1 21539.668,E2 21539.668} C_VEL
LIN {X 0,Y 452.916,Z 409.461,A -85,B 0,C 180,E1 21539.121,E2 21539.121} C_VEL
LIN {X 0,Y 450.23,Z 521.127,A -85,B 0,C 180,E1 21536.98,E2 21536.98} C_VEL
LIN {X 0,Y 449.019,Z 588.522,A -85,B 0,C 180,E1 21535.768,E2 21535.768} C_VEL
LIN {X 0,Y 448.187,Z 607.724,A -85,B 0,C 180,E1 21535.19,E2 21535.19} C_VEL
LIN {X 0,Y 447.127,Z 626.894,A -85,B 0,C 180,E1 21534.358,E2 21534.358} C_VEL
LIN {X 0,Y 446.057,Z 643.98,A -85,B 0,C 180,E1 21533.376,E2 21533.376} C_VEL
LIN {X 0,Y 444.879,Z 661.425,A -85,B 0,C 180,E1 21532.115,E2 21532.115} C_VEL
LIN {X 0,Y 443.721,Z 677.952,A -85,B 0,C 180,E1 21530.637,E2 21530.637} C_VEL
LIN {X 0,Y 442.701,Z 693.127,A -85,B 0,C 180,E1 21528.98,E2 21528.98} C_VEL
LIN {X 0,Y 441.858,Z 706.407,A -85,B 0,C 180,E1 21527.244,E2 21527.244} C_VEL
LIN {X 0,Y 441.172,Z 719.139,A -85,B 0,C 180,E1 21525.243,E2 21525.243} C_VEL
LIN {X 0,Y 440.711,Z 730.286,A -85,B 0,C 180,E1 21523.114,E2 21523.114} C_VEL
LIN {X 0,Y 440.459,Z 739.826,A -85,B 0,C 180,E1 21520.861,E2 21520.861} C_VEL
LIN {X 0,Y 440.382,Z 747.305,A -85,B 0,C 180,E1 21518.619,E2 21518.619} C_VEL
LIN {X 0,Y 440.396,Z 752.935,A -85,B 0,C 180,E1 21516.388,E2 21516.388} C_VEL
LIN {X 0,Y 440.469,Z 756.851,A -85,B 0,C 180,E1 21514.167,E2 21514.167} C_VEL
LIN {X 0,Y 440.53,Z 759.226,A -85,B 0,C 180,E1 21511.822,E2 21511.822} C_VEL
LIN {X 0,Y 440.532,Z 759.828,A -85,B 0,C 180,E1 21509.481,E2 21509.481} C_VEL
LIN {X 0,Y 440.472,Z 758.666,A -85,B 0,C 180,E1 21507.138,E2 21507.138} C_VEL
LIN {X 0,Y 440.38,Z 755.723,A -85,B 0,C 180,E1 21504.79,E2 21504.79} C_VEL
LIN {X 0,Y 440.315,Z 750.935,A -85,B 0,C 180,E1 21502.433,E2 21502.433} C_VEL
LIN {X 0,Y 440.344,Z 744.608,A -85,B 0,C 180,E1 21500.196,E2 21500.196} C_VEL
LIN {X 0,Y 440.52,Z 736.364,A -85,B 0,C 180,E1 21497.948,E2 21497.948} C_VEL
LIN {X 0,Y 440.903,Z 726.622,A -85,B 0,C 180,E1 21495.824,E2 21495.824} C_VEL
LIN {X 0,Y 441.498,Z 715.193,A -85,B 0,C 180,E1 21493.789,E2 21493.789} C_VEL
LIN {X 0,Y 442.292,Z 702.785,A -85,B 0,C 180,E1 21491.96,E2 21491.96} C_VEL
LIN {X 0,Y 443.28,Z 688.663,A -85,B 0,C 180,E1 21490.225,E2 21490.225} C_VEL
LIN {X 0,Y 444.428,Z 672.885,A -85,B 0,C 180,E1 21488.627,E2 21488.627} C_VEL
LIN {X 0,Y 445.591,Z 656.786,A -85,B 0,C 180,E1 21487.299,E2 21487.299} C_VEL
LIN {X 0,Y 446.729,Z 639.831,A -85,B 0,C 180,E1 21486.173,E2 21486.173} C_VEL
LIN {X 0,Y 447.783,Z 622.024,A -85,B 0,C 180,E1 21485.251,E2 21485.251} C_VEL
LIN {X 0,Y 448.687,Z 603.553,A -85,B 0,C 180,E1 21484.545,E2 21484.545} C_VEL
LIN {X 0,Y 449.364,Z 584.063,A -85,B 0,C 180,E1 21484.054,E2 21484.054} C_VEL
LIN {X 0,Y 452.237,Z 407.37,A -85,B 0,C 180,E1 21480.991,E2 21480.991} C_VEL
LIN {X 0,Y 449.959,Z 387.762,A -85,B 0,C 180,E1 21480.48,E2 21480.48} C_VEL
LIN {X 0,Y 453.454,Z 343.32,A -85,B 0,C 180,E1 21476.397,E2 21476.397} C_VEL
LIN {X 0,Y 454.158,Z 333.046,A -85,B 0,C 180,E1 21475.426,E2 21475.426} C_VEL
LIN {X 0,Y 446.112,Z 310.03,A -85,B 0,C 180,E1 21472.439,E2 21472.439} C_VEL
LIN {X 0,Y 441.126,Z 295.849,A -85,B 0,C 180,E1 21470.481,E2 21470.481} C_VEL
LIN {X 0,Y 441.12,Z 295.849,A -85,B 0,C 180,E1 21466.803,E2 21466.803} C_VEL
LIN {X 0,Y 441.129,Z 295.846,A -85,B 0,C 180,E1 21463.129,E2 21463.129} C_VEL
LIN {X 0,Y 441.166,Z 295.846,A -85,B 0,C 180,E1 21459.559,E2 21459.559} C_VEL
LIN {X 0,Y 441.168,Z 295.847,A -85,B 0,C 180,E1 21455.772,E2 21455.772} C_VEL
LIN {X 0,Y 441.152,Z 295.845,A -85,B 0,C 180,E1 21452.031,E2 21452.031} C_VEL
LIN {X 0,Y 441.129,Z 295.845,A -85,B 0,C 180,E1 21448.425,E2 21448.425} C_VEL
LIN {X 0,Y 441.125,Z 295.844,A -85,B 0,C 180,E1 21444.648,E2 21444.648} C_VEL
LIN {X 0,Y 441.128,Z 295.844,A -85,B 0,C 180,E1 21440.847,E2 21440.847} C_VEL
LIN {X 0,Y 441.155,Z 295.844,A -85,B 0,C 180,E1 21437.273,E2 21437.273} C_VEL
LIN {X 0,Y 441.18,Z 295.844,A -85,B 0,C 180,E1 21433.534,E2 21433.534} C_VEL
LIN {X 0,Y 441.17,Z 295.845,A -85,B 0,C 180,E1 21429.788,E2 21429.788} C_VEL
LIN {X 0,Y 441.136,Z 295.844,A -85,B 0,C 180,E1 21426.248,E2 21426.248} C_VEL
LIN {X 0,Y 441.129,Z 295.844,A -85,B 0,C 180,E1 21422.6,E2 21422.6} C_VEL
LIN {X 0,Y 441.141,Z 295.843,A -85,B 0,C 180,E1 21418.963,E2 21418.963} C_VEL
LIN {X 0,Y 441.168,Z 295.843,A -85,B 0,C 180,E1 21415.322,E2 21415.322} C_VEL
LIN {X 0,Y 441.183,Z 295.845,A -85,B 0,C 180,E1 21411.662,E2 21411.662} C_VEL
LIN {X 0,Y 441.155,Z 295.844,A -85,B 0,C 180,E1 21407.967,E2 21407.967} C_VEL
LIN {X 0,Y 441.136,Z 295.843,A -85,B 0,C 180,E1 21404.355,E2 21404.355} C_VEL
LIN {X 0,Y 441.137,Z 295.843,A -85,B 0,C 180,E1 21400.538,E2 21400.538} C_VEL
LIN {X 0,Y 441.15,Z 295.842,A -85,B 0,C 180,E1 21396.917,E2 21396.917} C_VEL
LIN {X 0,Y 441.178,Z 295.842,A -85,B 0,C 180,E1 21393.242,E2 21393.242} C_VEL
LIN {X 0,Y 441.196,Z 295.842,A -85,B 0,C 180,E1 21389.446,E2 21389.446} C_VEL
LIN {X 0,Y 441.18,Z 295.844,A -85,B 0,C 180,E1 21385.648,E2 21385.648} C_VEL
LIN {X 0,Y 441.156,Z 295.843,A -85,B 0,C 180,E1 21381.944,E2 21381.944} C_VEL
LIN {X 0,Y 441.143,Z 295.842,A -85,B 0,C 180,E1 21378.391,E2 21378.391} C_VEL
LIN {X 0,Y 441.147,Z 295.842,A -85,B 0,C 180,E1 21374.632,E2 21374.632} C_VEL
LIN {X 0,Y 441.164,Z 295.841,A -85,B 0,C 180,E1 21370.918,E2 21370.918} C_VEL
LIN {X 0,Y 441.189,Z 295.841,A -85,B 0,C 180,E1 21367.234,E2 21367.234} C_VEL
LIN {X 0,Y 441.193,Z 295.843,A -85,B 0,C 180,E1 21363.414,E2 21363.414} C_VEL
LIN {X 0,Y 441.169,Z 295.843,A -85,B 0,C 180,E1 21359.757,E2 21359.757} C_VEL
LIN {X 0,Y 441.151,Z 295.842,A -85,B 0,C 180,E1 21356.083,E2 21356.083} C_VEL
LIN {X 0,Y 441.15,Z 295.841,A -85,B 0,C 180,E1 21352.38,E2 21352.38} C_VEL
LIN {X 0,Y 441.16,Z 295.84,A -85,B 0,C 180,E1 21348.682,E2 21348.682} C_VEL
LIN {X 0,Y 441.182,Z 295.84,A -85,B 0,C 180,E1 21344.972,E2 21344.972} C_VEL
LIN {X 0,Y 441.195,Z 295.841,A -85,B 0,C 180,E1 21341.238,E2 21341.238} C_VEL
LIN {X 0,Y 441.193,Z 295.844,A -85,B 0,C 180,E1 21337.421,E2 21337.421} C_VEL
LIN {X 0,Y 441.155,Z 295.841,A -85,B 0,C 180,E1 21336.473,E2 21336.473} C_VEL
LIN {X 0,Y 440.142,Z 295.974,A -85,B 0,C 180,E1 21335.473,E2 21335.473} C_VEL
LIN {X 0,Y 433.631,Z 296.78,A -85,B 0,C 180,E1 21332.582,E2 21332.582} C_VEL
LIN {X 0,Y 433.219,Z 296.831,A -85,B 0,C 180,E1 21331.919,E2 21331.919} C_VEL
LIN {X 0,Y 433.214,Z 296.83,A -85,B 0,C 180,E1 21328.147,E2 21328.147} C_VEL
LIN {X 0,Y 433.215,Z 296.83,A -85,B 0,C 180,E1 21324.303,E2 21324.303} C_VEL
LIN {X 0,Y 433.226,Z 296.829,A -85,B 0,C 180,E1 21320.568,E2 21320.568} C_VEL
LIN {X 0,Y 433.242,Z 296.828,A -85,B 0,C 180,E1 21316.792,E2 21316.792} C_VEL
LIN {X 0,Y 433.26,Z 296.829,A -85,B 0,C 180,E1 21313.095,E2 21313.095} C_VEL
LIN {X 0,Y 433.256,Z 296.832,A -85,B 0,C 180,E1 21309.323,E2 21309.323} C_VEL
LIN {X 0,Y 433.235,Z 296.832,A -85,B 0,C 180,E1 21305.599,E2 21305.599} C_VEL
LIN {X 0,Y 433.227,Z 296.83,A -85,B 0,C 180,E1 21301.833,E2 21301.833} C_VEL
LIN {X 0,Y 433.221,Z 296.829,A -85,B 0,C 180,E1 21298.093,E2 21298.093} C_VEL
LIN {X 0,Y 433.226,Z 296.828,A -85,B 0,C 180,E1 21294.273,E2 21294.273} C_VEL
LIN {X 0,Y 433.243,Z 296.827,A -85,B 0,C 180,E1 21290.604,E2 21290.604} C_VEL
LIN {X 0,Y 433.256,Z 296.827,A -85,B 0,C 180,E1 21286.82,E2 21286.82} C_VEL
LIN {X 0,Y 433.261,Z 296.832,A -85,B 0,C 180,E1 21282.982,E2 21282.982} C_VEL
LIN {X 0,Y 433.264,Z 296.831,A -85,B 0,C 180,E1 21279.158,E2 21279.158} C_VEL
LIN {X 0,Y 433.245,Z 296.832,A -85,B 0,C 180,E1 21275.396,E2 21275.396} C_VEL
LIN {X 0,Y 433.264,Z 296.977,A -85,B 0,C 180,E1 21274.525,E2 21274.525} C_VEL
LIN {X 0,Y 438.822,Z 317.267,A -85,B 0,C 180,E1 21271.048,E2 21271.048} C_VEL
LIN {X 0,Y 441.155,Z 326.982,A -85,B 0,C 180,E1 21269.457,E2 21269.457} C_VEL
LIN {X 0,Y 439.122,Z 355.525,A -85,B 0,C 180,E1 21265.487,E2 21265.487} C_VEL
LIN {X 0,Y 437.279,Z 384.824,A -85,B 0,C 180,E1 21261.466,E2 21261.466} C_VEL
LIN {X 0,Y 436.284,Z 403.334,A -85,B 0,C 180,E1 21258.997,E2 21258.997} C_VEL
LIN {X 0,Y 439.292,Z 424.581,A -85,B 0,C 180,E1 21258.394,E2 21258.394} C_VEL
LIN {X 0,Y 437.184,Z 525.188,A -85,B 0,C 180,E1 21256.315,E2 21256.315} C_VEL
LIN {X 0,Y 436.803,Z 540.45,A -85,B 0,C 180,E1 21255.77,E2 21255.77} C_VEL
LIN {X 0,Y 436.256,Z 556.321,A -85,B 0,C 180,E1 21254.94,E2 21254.94} C_VEL
LIN {X 0,Y 435.607,Z 571.53,A -85,B 0,C 180,E1 21253.848,E2 21253.848} C_VEL
LIN {X 0,Y 434.985,Z 584.692,A -85,B 0,C 180,E1 21252.611,E2 21252.611} C_VEL
LIN {X 0,Y 434.426,Z 595.961,A -85,B 0,C 180,E1 21251.28,E2 21251.28} C_VEL
LIN {X 0,Y 433.9,Z 606.708,A -85,B 0,C 180,E1 21249.682,E2 21249.682} C_VEL
LIN {X 0,Y 433.481,Z 615.735,A -85,B 0,C 180,E1 21247.953,E2 21247.953} C_VEL
LIN {X 0,Y 433.212,Z 622.662,A -85,B 0,C 180,E1 21246.225,E2 21246.225} C_VEL
LIN {X 0,Y 433.054,Z 628.177,A -85,B 0,C 180,E1 21244.368,E2 21244.368} C_VEL
LIN {X 0,Y 432.982,Z 632.007,A -85,B 0,C 180,E1 21242.38,E2 21242.38} C_VEL
LIN {X 0,Y 433.008,Z 633.875,A -85,B 0,C 180,E1 21240.527,E2 21240.527} C_VEL
LIN {X 0,Y 433.105,Z 634.042,A -85,B 0,C 180,E1 21238.543,E2 21238.543} C_VEL
LIN {X 0,Y 433.275,Z 632.468,A -85,B 0,C 180,E1 21236.691,E2 21236.691} C_VEL
LIN {X 0,Y 433.57,Z 628.92,A -85,B 0,C 180,E1 21234.705,E2 21234.705} C_VEL
LIN {X 0,Y 433.95,Z 623.654,A -85,B 0,C 180,E1 21232.851,E2 21232.851} C_VEL
LIN {X 0,Y 434.456,Z 616.922,A -85,B 0,C 180,E1 21231.128,E2 21231.128} C_VEL
LIN {X 0,Y 435.111,Z 608.006,A -85,B 0,C 180,E1 21229.405,E2 21229.405} C_VEL
LIN {X 0,Y 435.871,Z 597.359,A -85,B 0,C 180,E1 21227.815,E2 21227.815} C_VEL
LIN {X 0,Y 436.647,Z 585.843,A -85,B 0,C 180,E1 21226.452,E2 21226.452} C_VEL
LIN {X 0,Y 437.477,Z 572.712,A -85,B 0,C 180,E1 21225.228,E2 21225.228} C_VEL
LIN {X 0,Y 438.259,Z 558.052,A -85,B 0,C 180,E1 21224.178,E2 21224.178} C_VEL
LIN {X 0,Y 438.925,Z 542.942,A -85,B 0,C 180,E1 21223.369,E2 21223.369} C_VEL
LIN {X 0,Y 439.479,Z 527.039,A -85,B 0,C 180,E1 21222.765,E2 21222.765} C_VEL
LIN {X 0,Y 443.986,Z 435.232,A -85,B 0,C 180,E1 21220.279,E2 21220.279} C_VEL
LIN {X 0,Y 444.362,Z 425.853,A -85,B 0,C 180,E1 21219.999,E2 21219.999} C_VEL
LIN {X 0,Y 440.838,Z 406.02,A -85,B 0,C 180,E1 21219.022,E2 21219.022} C_VEL
LIN {X 0,Y 440.291,Z 402.972,A -85,B 0,C 180,E1 21218.832,E2 21218.832} C_VEL
LIN {X 0,Y 443.172,Z 376.544,A -85,B 0,C 180,E1 21214.901,E2 21214.901} C_VEL
LIN {X 0,Y 446.822,Z 351.217,A -85,B 0,C 180,E1 21210.948,E2 21210.948} C_VEL
LIN {X 0,Y 448.716,Z 339.948,A -85,B 0,C 180,E1 21209.081,E2 21209.081} C_VEL
LIN {X 0,Y 446.753,Z 330.841,A -85,B 0,C 180,E1 21206.829,E2 21206.829} C_VEL
LIN {X 0,Y 444.803,Z 323.834,A -85,B 0,C 180,E1 21204.685,E2 21204.685} C_VEL
LIN {X 0,Y 443.18,Z 318.46,A -85,B 0,C 180,E1 21202.576,E2 21202.576} C_VEL
LIN {X 0,Y 441.846,Z 314.867,A -85,B 0,C 180,E1 21200.504,E2 21200.504} C_VEL
LIN {X 0,Y 440.97,Z 312.737,A -85,B 0,C 180,E1 21198.018,E2 21198.018} C_VEL
LIN {X 0,Y 441.068,Z 312.628,A -85,B 0,C 180,E1 21196.077,E2 21196.077} C_VEL
LIN {X 0,Y 441.915,Z 314.656,A -85,B 0,C 180,E1 21193.799,E2 21193.799} C_VEL
LIN {X 0,Y 442.921,Z 316.305,A -85,B 0,C 180,E1 21192.614,E2 21192.614} C_VEL
LIN {X 0,Y 444.674,Z 320.785,A -85,B 0,C 180,E1 21190.699,E2 21190.699} C_VEL
LIN {X 0,Y 446.937,Z 326.587,A -85,B 0,C 180,E1 21188.873,E2 21188.873} C_VEL
LIN {X 0,Y 449.516,Z 334.36,A -85,B 0,C 180,E1 21187.009,E2 21187.009} C_VEL
LIN {X 0,Y 451.515,Z 342.019,A -85,B 0,C 180,E1 21185.543,E2 21185.543} C_VEL
LIN {X 0,Y 446.78,Z 369.707,A -85,B 0,C 180,E1 21182.466,E2 21182.466} C_VEL
LIN {X 0,Y 444.151,Z 391.658,A -85,B 0,C 180,E1 21180.22,E2 21180.22} C_VEL
LIN {X 0,Y 446.006,Z 409.998,A -85,B 0,C 180,E1 21179.63,E2 21179.63} C_VEL
LIN {X 0,Y 443.064,Z 518.617,A -85,B 0,C 180,E1 21177.471,E2 21177.471} C_VEL
LIN {X 0,Y 441.647,Z 588.028,A -85,B 0,C 180,E1 21176.176,E2 21176.176} C_VEL
LIN {X 0,Y 440.725,Z 607.534,A -85,B 0,C 180,E1 21175.571,E2 21175.571} C_VEL
LIN {X 0,Y 439.604,Z 626.149,A -85,B 0,C 180,E1 21174.741,E2 21174.741} C_VEL
LIN {X 0,Y 438.434,Z 643.565,A -85,B 0,C 180,E1 21173.717,E2 21173.717} C_VEL
LIN {X 0,Y 437.191,Z 660.615,A -85,B 0,C 180,E1 21172.454,E2 21172.454} C_VEL
LIN {X 0,Y 435.956,Z 676.922,A -85,B 0,C 180,E1 21170.965,E2 21170.965} C_VEL
LIN {X 0,Y 434.855,Z 692.177,A -85,B 0,C 180,E1 21169.267,E2 21169.267} C_VEL
LIN {X 0,Y 433.931,Z 705.879,A -85,B 0,C 180,E1 21167.431,E2 21167.431} C_VEL
LIN {X 0,Y 433.21,Z 718.515,A -85,B 0,C 180,E1 21165.393,E2 21165.393} C_VEL
LIN {X 0,Y 432.73,Z 729.581,A -85,B 0,C 180,E1 21163.224,E2 21163.224} C_VEL
LIN {X 0,Y 432.487,Z 738.544,A -85,B 0,C 180,E1 21161.064,E2 21161.064} C_VEL
LIN {X 0,Y 432.419,Z 746.072,A -85,B 0,C 180,E1 21158.779,E2 21158.779} C_VEL
LIN {X 0,Y 432.445,Z 751.741,A -85,B 0,C 180,E1 21156.506,E2 21156.506} C_VEL
LIN {X 0,Y 432.532,Z 755.689,A -85,B 0,C 180,E1 21154.243,E2 21154.243} C_VEL
LIN {X 0,Y 432.608,Z 758.088,A -85,B 0,C 180,E1 21151.855,E2 21151.855} C_VEL
LIN {X 0,Y 432.612,Z 758.7,A -85,B 0,C 180,E1 21149.471,E2 21149.471} C_VEL
LIN {X 0,Y 432.542,Z 757.531,A -85,B 0,C 180,E1 21147.086,E2 21147.086} C_VEL
LIN {X 0,Y 432.43,Z 754.567,A -85,B 0,C 180,E1 21144.694,E2 21144.694} C_VEL
LIN {X 0,Y 432.353,Z 749.741,A -85,B 0,C 180,E1 21142.293,E2 21142.293} C_VEL
LIN {X 0,Y 432.377,Z 743.358,A -85,B 0,C 180,E1 21140.013,E2 21140.013} C_VEL
LIN {X 0,Y 432.555,Z 735.038,A -85,B 0,C 180,E1 21137.723,E2 21137.723} C_VEL
LIN {X 0,Y 432.966,Z 725.201,A -85,B 0,C 180,E1 21135.559,E2 21135.559} C_VEL
LIN {X 0,Y 433.589,Z 713.901,A -85,B 0,C 180,E1 21133.524,E2 21133.524} C_VEL
LIN {X 0,Y 434.484,Z 700.788,A -85,B 0,C 180,E1 21131.574,E2 21131.574} C_VEL
LIN {X 0,Y 435.556,Z 686.204,A -85,B 0,C 180,E1 21129.79,E2 21129.79} C_VEL
LIN {X 0,Y 436.732,Z 670.715,A -85,B 0,C 180,E1 21128.231,E2 21128.231} C_VEL
LIN {X 0,Y 437.965,Z 654.273,A -85,B 0,C 180,E1 21126.88,E2 21126.88} C_VEL
LIN {X 0,Y 439.172,Z 636.896,A -85,B 0,C 180,E1 21125.737,E2 21125.737} C_VEL
LIN {X 0,Y 440.303,Z 618.447,A -85,B 0,C 180,E1 21124.801,E2 21124.801} C_VEL
LIN {X 0,Y 441.243,Z 599.881,A -85,B 0,C 180,E1 21124.119,E2 21124.119} C_VEL
LIN {X 0,Y 441.847,Z 580.861,A -85,B 0,C 180,E1 21123.664,E2 21123.664} C_VEL
LIN {X 0,Y 444.894,Z 408.654,A -85,B 0,C 180,E1 21120.619,E2 21120.619} C_VEL
LIN {X 0,Y 442.523,Z 387.601,A -85,B 0,C 180,E1 21120.045,E2 21120.045} C_VEL
LIN {X 0,Y 446.125,Z 344.617,A -85,B 0,C 180,E1 21116.023,E2 21116.023} C_VEL
LIN {X 0,Y 446.892,Z 335.997,A -85,B 0,C 180,E1 21115.198,E2 21115.198} C_VEL
LIN {X 0,Y 438.454,Z 311.772,A -85,B 0,C 180,E1 21111.998,E2 21111.998} C_VEL
LIN {X 0,Y 433.232,Z 296.834,A -85,B 0,C 180,E1 21109.875,E2 21109.875} C_VEL
LIN {X 0,Y 433.203,Z 296.838,A -85,B 0,C 180,E1 21106.18,E2 21106.18} C_VEL
LIN {X 0,Y 433.184,Z 296.835,A -85,B 0,C 180,E1 21102.556,E2 21102.556} C_VEL
LIN {X 0,Y 433.182,Z 296.834,A -85,B 0,C 180,E1 21098.727,E2 21098.727} C_VEL
LIN {X 0,Y 433.186,Z 296.834,A -85,B 0,C 180,E1 21094.921,E2 21094.921} C_VEL
LIN {X 0,Y 433.207,Z 296.833,A -85,B 0,C 180,E1 21091.287,E2 21091.287} C_VEL
LIN {X 0,Y 433.237,Z 296.834,A -85,B 0,C 180,E1 21087.6,E2 21087.6} C_VEL
LIN {X 0,Y 433.232,Z 296.834,A -85,B 0,C 180,E1 21083.823,E2 21083.823} C_VEL
LIN {X 0,Y 433.197,Z 296.833,A -85,B 0,C 180,E1 21080.257,E2 21080.257} C_VEL
LIN {X 0,Y 433.188,Z 296.833,A -85,B 0,C 180,E1 21076.633,E2 21076.633} C_VEL
LIN {X 0,Y 433.194,Z 296.833,A -85,B 0,C 180,E1 21072.939,E2 21072.939} C_VEL
LIN {X 0,Y 433.22,Z 296.832,A -85,B 0,C 180,E1 21069.299,E2 21069.299} C_VEL
LIN {X 0,Y 433.24,Z 296.834,A -85,B 0,C 180,E1 21065.697,E2 21065.697} C_VEL
LIN {X 0,Y 433.226,Z 296.833,A -85,B 0,C 180,E1 21061.853,E2 21061.853} C_VEL
LIN {X 0,Y 433.198,Z 296.833,A -85,B 0,C 180,E1 21058.283,E2 21058.283} C_VEL
LIN {X 0,Y 433.192,Z 296.833,A -85,B 0,C 180,E1 21054.572,E2 21054.572} C_VEL
LIN {X 0,Y 433.2,Z 296.832,A -85,B 0,C 180,E1 21050.838,E2 21050.838} C_VEL
LIN {X 0,Y 433.226,Z 296.831,A -85,B 0,C 180,E1 21047.201,E2 21047.201} C_VEL
LIN {X 0,Y 433.248,Z 296.833,A -85,B 0,C 180,E1 21043.512,E2 21043.512} C_VEL
LIN {X 0,Y 433.233,Z 296.833,A -85,B 0,C 180,E1 21039.748,E2 21039.748} C_VEL
LIN {X 0,Y 433.205,Z 296.832,A -85,B 0,C 180,E1 21036.18,E2 21036.18} C_VEL
LIN {X 0,Y 433.201,Z 296.832,A -85,B 0,C 180,E1 21032.409,E2 21032.409} C_VEL
LIN {X 0,Y 433.202,Z 296.831,A -85,B 0,C 180,E1 21028.562,E2 21028.562} C_VEL
LIN {X 0,Y 433.218,Z 296.831,A -85,B 0,C 180,E1 21024.925,E2 21024.925} C_VEL
LIN {X 0,Y 433.252,Z 296.829,A -85,B 0,C 180,E1 21021.262,E2 21021.262} C_VEL
LIN {X 0,Y 433.242,Z 296.833,A -85,B 0,C 180,E1 21017.603,E2 21017.603} C_VEL
LIN {X 0,Y 433.224,Z 296.833,A -85,B 0,C 180,E1 21013.817,E2 21013.817} C_VEL
LIN {X 0,Y 433.207,Z 296.832,A -85,B 0,C 180,E1 21010.19,E2 21010.19} C_VEL
LIN {X 0,Y 433.206,Z 296.831,A -85,B 0,C 180,E1 21006.346,E2 21006.346} C_VEL
LIN {X 0,Y 433.211,Z 296.83,A -85,B 0,C 180,E1 21002.53,E2 21002.53} C_VEL
LIN {X 0,Y 433.226,Z 296.829,A -85,B 0,C 180,E1 20998.838,E2 20998.838} C_VEL
LIN {X 0,Y 433.247,Z 296.829,A -85,B 0,C 180,E1 20995.127,E2 20995.127} C_VEL
LIN {X 0,Y 433.261,Z 296.831,A -85,B 0,C 180,E1 20991.383,E2 20991.383} C_VEL
LIN {X 0,Y 433.24,Z 296.833,A -85,B 0,C 180,E1 20987.596,E2 20987.596} C_VEL
LIN {X 0,Y 433.22,Z 296.832,A -85,B 0,C 180,E1 20983.887,E2 20983.887} C_VEL
LIN {X 0,Y 433.211,Z 296.831,A -85,B 0,C 180,E1 20980.236,E2 20980.236} C_VEL
LIN {X 0,Y 433.216,Z 296.83,A -85,B 0,C 180,E1 20976.478,E2 20976.478} C_VEL
LIN {X 0,Y 433.233,Z 296.829,A -85,B 0,C 180,E1 20972.777,E2 20972.777} C_VEL
LIN {X 0,Y 433.219,Z 296.831,A -85,B 0,C 180,E1 20971.919,E2 20971.919} C_VEL
LIN {X 0,Y 432.261,Z 296.959,A -85,B 0,C 180,E1 20970.9,E2 20970.9} C_VEL
LIN {X 0,Y 425.748,Z 297.774,A -85,B 0,C 180,E1 20967.956,E2 20967.956} C_VEL
LIN {X 0,Y 425.314,Z 297.82,A -85,B 0,C 180,E1 20967.281,E2 20967.281} C_VEL
LIN {X 0,Y 425.315,Z 297.822,A -85,B 0,C 180,E1 20963.384,E2 20963.384} C_VEL
LIN {X 0,Y 425.299,Z 297.821,A -85,B 0,C 180,E1 20959.57,E2 20959.57} C_VEL
LIN {X 0,Y 425.282,Z 297.82,A -85,B 0,C 180,E1 20955.846,E2 20955.846} C_VEL
LIN {X 0,Y 425.28,Z 297.819,A -85,B 0,C 180,E1 20952.061,E2 20952.061} C_VEL
LIN {X 0,Y 425.28,Z 297.818,A -85,B 0,C 180,E1 20948.193,E2 20948.193} C_VEL
LIN {X 0,Y 425.286,Z 297.818,A -85,B 0,C 180,E1 20944.367,E2 20944.367} C_VEL
LIN {X 0,Y 425.299,Z 297.816,A -85,B 0,C 180,E1 20940.57,E2 20940.57} C_VEL
LIN {X 0,Y 425.311,Z 297.816,A -85,B 0,C 180,E1 20936.786,E2 20936.786} C_VEL
LIN {X 0,Y 425.322,Z 297.817,A -85,B 0,C 180,E1 20932.999,E2 20932.999} C_VEL
LIN {X 0,Y 425.325,Z 297.819,A -85,B 0,C 180,E1 20929.191,E2 20929.191} C_VEL
LIN {X 0,Y 425.311,Z 297.822,A -85,B 0,C 180,E1 20925.337,E2 20925.337} C_VEL
LIN {X 0,Y 425.301,Z 297.82,A -85,B 0,C 180,E1 20921.523,E2 20921.523} C_VEL
LIN {X 0,Y 425.289,Z 297.822,A -85,B 0,C 180,E1 20917.819,E2 20917.819} C_VEL
LIN {X 0,Y 425.329,Z 297.88,A -85,B 0,C 180,E1 20915.035,E2 20915.035} C_VEL
LIN {X 0,Y 430.938,Z 318.299,A -85,B 0,C 180,E1 20911.466,E2 20911.466} C_VEL
LIN {X 0,Y 433.598,Z 328.767,A -85,B 0,C 180,E1 20909.718,E2 20909.718} C_VEL
LIN {X 0,Y 431.486,Z 356.838,A -85,B 0,C 180,E1 20905.75,E2 20905.75} C_VEL
LIN {X 0,Y 429.571,Z 385.843,A -85,B 0,C 180,E1 20901.718,E2 20901.718} C_VEL
LIN {X 0,Y 428.586,Z 403.25,A -85,B 0,C 180,E1 20899.361,E2 20899.361} C_VEL
LIN {X 0,Y 431.692,Z 425.603,A -85,B 0,C 180,E1 20898.712,E2 20898.712} C_VEL
LIN {X 0,Y 429.449,Z 525.95,A -85,B 0,C 180,E1 20896.573,E2 20896.573} C_VEL
LIN {X 0,Y 429.03,Z 541.645,A -85,B 0,C 180,E1 20895.994,E2 20895.994} C_VEL
LIN {X 0,Y 428.464,Z 557.37,A -85,B 0,C 180,E1 20895.149,E2 20895.149} C_VEL
LIN {X 0,Y 427.805,Z 572.2,A -85,B 0,C 180,E1 20894.065,E2 20894.065} C_VEL
LIN {X 0,Y 427.144,Z 585.704,A -85,B 0,C 180,E1 20892.778,E2 20892.778} C_VEL
LIN {X 0,Y 426.588,Z 596.482,A -85,B 0,C 180,E1 20891.49,E2 20891.49} C_VEL
LIN {X 0,Y 426.032,Z 607.366,A -85,B 0,C 180,E1 20889.863,E2 20889.863} C_VEL
LIN {X 0,Y 425.589,Z 616.519,A -85,B 0,C 180,E1 20888.101,E2 20888.101} C_VEL
LIN {X 0,Y 425.305,Z 623.561,A -85,B 0,C 180,E1 20886.342,E2 20886.342} C_VEL
LIN {X 0,Y 425.137,Z 629.177,A -85,B 0,C 180,E1 20884.449,E2 20884.449} C_VEL
LIN {X 0,Y 425.065,Z 633.109,A -85,B 0,C 180,E1 20882.425,E2 20882.425} C_VEL
LIN {X 0,Y 425.096,Z 635.061,A -85,B 0,C 180,E1 20880.537,E2 20880.537} C_VEL
LIN {X 0,Y 425.207,Z 635.3,A -85,B 0,C 180,E1 20878.516,E2 20878.516} C_VEL
LIN {X 0,Y 425.403,Z 633.819,A -85,B 0,C 180,E1 20876.63,E2 20876.63} C_VEL
LIN {X 0,Y 425.73,Z 630.334,A -85,B 0,C 180,E1 20874.608,E2 20874.608} C_VEL
LIN {X 0,Y 426.15,Z 625.129,A -85,B 0,C 180,E1 20872.719,E2 20872.719} C_VEL
LIN {X 0,Y 426.704,Z 618.473,A -85,B 0,C 180,E1 20870.966,E2 20870.966} C_VEL
LIN {X 0,Y 427.42,Z 609.676,A -85,B 0,C 180,E1 20869.212,E2 20869.212} C_VEL
LIN {X 0,Y 428.175,Z 600.177,A -85,B 0,C 180,E1 20867.729,E2 20867.729} C_VEL
LIN {X 0,Y 429.055,Z 588.199,A -85,B 0,C 180,E1 20866.248,E2 20866.248} C_VEL
LIN {X 0,Y 430.008,Z 574.226,A -85,B 0,C 180,E1 20864.903,E2 20864.903} C_VEL
LIN {X 0,Y 430.925,Z 558.74,A -85,B 0,C 180,E1 20863.763,E2 20863.763} C_VEL
LIN {X 0,Y 431.704,Z 542.656,A -85,B 0,C 180,E1 20862.892,E2 20862.892} C_VEL
LIN {X 0,Y 432.304,Z 526.129,A -85,B 0,C 180,E1 20862.275,E2 20862.275} C_VEL
LIN {X 0,Y 437.38,Z 433.505,A -85,B 0,C 180,E1 20859.661,E2 20859.661} C_VEL
LIN {X 0,Y 437.574,Z 427.092,A -85,B 0,C 180,E1 20859.453,E2 20859.453} C_VEL
LIN {X 0,Y 434.24,Z 407.95,A -85,B 0,C 180,E1 20858.459,E2 20858.459} C_VEL
LIN {X 0,Y 433.301,Z 402.929,A -85,B 0,C 180,E1 20858.154,E2 20858.154} C_VEL
LIN {X 0,Y 436.567,Z 376.158,A -85,B 0,C 180,E1 20854.058,E2 20854.058} C_VEL
LIN {X 0,Y 440.645,Z 351.307,A -85,B 0,C 180,E1 20850.052,E2 20850.052} C_VEL
LIN {X 0,Y 442.075,Z 343.72,A -85,B 0,C 180,E1 20848.754,E2 20848.754} C_VEL
LIN {X 0,Y 440.281,Z 334.902,A -85,B 0,C 180,E1 20846.455,E2 20846.455} C_VEL
LIN {X 0,Y 438.524,Z 328.282,A -85,B 0,C 180,E1 20844.288,E2 20844.288} C_VEL
LIN {X 0,Y 437.06,Z 323.391,A -85,B 0,C 180,E1 20842.185,E2 20842.185} C_VEL
LIN {X 0,Y 436.156,Z 320.453,A -85,B 0,C 180,E1 20840.378,E2 20840.378} C_VEL
LIN {X 0,Y 435.477,Z 318.423,A -85,B 0,C 180,E1 20837.674,E2 20837.674} C_VEL
LIN {X 0,Y 435.715,Z 318.721,A -85,B 0,C 180,E1 20835.723,E2 20835.723} C_VEL
LIN {X 0,Y 436.877,Z 321.171,A -85,B 0,C 180,E1 20833.297,E2 20833.297} C_VEL
LIN {X 0,Y 437.532,Z 322.782,A -85,B 0,C 180,E1 20832.389,E2 20832.389} C_VEL
LIN {X 0,Y 439.022,Z 326.395,A -85,B 0,C 180,E1 20830.817,E2 20830.817} C_VEL
LIN {X 0,Y 441.123,Z 332.142,A -85,B 0,C 180,E1 20828.971,E2 20828.971} C_VEL
LIN {X 0,Y 443.431,Z 339.429,A -85,B 0,C 180,E1 20827.179,E2 20827.179} C_VEL
LIN {X 0,Y 444.946,Z 345.512,A -85,B 0,C 180,E1 20825.958,E2 20825.958} C_VEL
LIN {X 0,Y 440.04,Z 371.559,A -85,B 0,C 180,E1 20822.97,E2 20822.97} C_VEL
LIN {X 0,Y 437.314,Z 392.041,A -85,B 0,C 180,E1 20820.811,E2 20820.811} C_VEL
LIN {X 0,Y 439.235,Z 410.302,A -85,B 0,C 180,E1 20820.181,E2 20820.181} C_VEL
LIN {X 0,Y 435.988,Z 515.953,A -85,B 0,C 180,E1 20817.995,E2 20817.995} C_VEL
LIN {X 0,Y 434.346,Z 587.191,A -85,B 0,C 180,E1 20816.618,E2 20816.618} C_VEL
LIN {X 0,Y 433.352,Z 606.654,A -85,B 0,C 180,E1 20816.002,E2 20816.002} C_VEL
LIN {X 0,Y 432.154,Z 625.142,A -85,B 0,C 180,E1 20815.16,E2 20815.16} C_VEL
LIN {X 0,Y 430.882,Z 642.733,A -85,B 0,C 180,E1 20814.106,E2 20814.106} C_VEL
LIN {X 0,Y 429.527,Z 659.92,A -85,B 0,C 180,E1 20812.805,E2 20812.805} C_VEL
LIN {X 0,Y 428.211,Z 675.985,A -85,B 0,C 180,E1 20811.304,E2 20811.304} C_VEL
LIN {X 0,Y 427.021,Z 691.295,A -85,B 0,C 180,E1 20809.563,E2 20809.563} C_VEL
LIN {X 0,Y 426.022,Z 705.181,A -85,B 0,C 180,E1 20807.659,E2 20807.659} C_VEL
LIN {X 0,Y 425.25,Z 717.933,A -85,B 0,C 180,E1 20805.549,E2 20805.549} C_VEL
LIN {X 0,Y 424.752,Z 728.909,A -85,B 0,C 180,E1 20803.339,E2 20803.339} C_VEL
LIN {X 0,Y 424.505,Z 737.79,A -85,B 0,C 180,E1 20801.137,E2 20801.137} C_VEL
LIN {X 0,Y 424.45,Z 745.245,A -85,B 0,C 180,E1 20798.809,E2 20798.809} C_VEL
LIN {X 0,Y 424.495,Z 750.84,A -85,B 0,C 180,E1 20796.493,E2 20796.493} C_VEL
LIN {X 0,Y 424.601,Z 754.713,A -85,B 0,C 180,E1 20794.187,E2 20794.187} C_VEL
LIN {X 0,Y 424.686,Z 756.945,A -85,B 0,C 180,E1 20791.89,E2 20791.89} C_VEL
LIN {X 0,Y 424.694,Z 757.558,A -85,B 0,C 180,E1 20789.461,E2 20789.461} C_VEL
LIN {X 0,Y 424.615,Z 756.376,A -85,B 0,C 180,E1 20787.032,E2 20787.032} C_VEL
LIN {X 0,Y 424.484,Z 753.383,A -85,B 0,C 180,E1 20784.595,E2 20784.595} C_VEL
LIN {X 0,Y 424.396,Z 748.835,A -85,B 0,C 180,E1 20782.284,E2 20782.284} C_VEL
LIN {X 0,Y 424.405,Z 742.506,A -85,B 0,C 180,E1 20779.961,E2 20779.961} C_VEL
LIN {X 0,Y 424.577,Z 734.22,A -85,B 0,C 180,E1 20777.627,E2 20777.627} C_VEL
LIN {X 0,Y 425.001,Z 724.407,A -85,B 0,C 180,E1 20775.421,E2 20775.421} C_VEL
LIN {X 0,Y 425.648,Z 713.122,A -85,B 0,C 180,E1 20773.348,E2 20773.348} C_VEL
LIN {X 0,Y 426.576,Z 700.043,A -85,B 0,C 180,E1 20771.364,E2 20771.364} C_VEL
LIN {X 0,Y 427.698,Z 685.48,A -85,B 0,C 180,E1 20769.545,E2 20769.545} C_VEL
LIN {X 0,Y 428.933,Z 669.985,A -85,B 0,C 180,E1 20767.959,E2 20767.959} C_VEL
LIN {X 0,Y 430.222,Z 653.53,A -85,B 0,C 180,E1 20766.585,E2 20766.585} C_VEL
LIN {X 0,Y 431.483,Z 636.128,A -85,B 0,C 180,E1 20765.422,E2 20765.422} C_VEL
LIN {X 0,Y 432.66,Z 617.645,A -85,B 0,C 180,E1 20764.471,E2 20764.471} C_VEL
LIN {X 0,Y 433.642,Z 599.194,A -85,B 0,C 180,E1 20763.783,E2 20763.783} C_VEL
LIN {X 0,Y 434.267,Z 580.077,A -85,B 0,C 180,E1 20763.319,E2 20763.319} C_VEL
LIN {X 0,Y 437.489,Z 410.791,A -85,B 0,C 180,E1 20760.26,E2 20760.26} C_VEL
LIN {X 0,Y 435.071,Z 387.741,A -85,B 0,C 180,E1 20759.631,E2 20759.631} C_VEL
LIN {X 0,Y 438.907,Z 344.746,A -85,B 0,C 180,E1 20755.531,E2 20755.531} C_VEL
LIN {X 0,Y 439.379,Z 338.285,A -85,B 0,C 180,E1 20754.895,E2 20754.895} C_VEL
LIN {X 0,Y 430.999,Z 314.169,A -85,B 0,C 180,E1 20751.64,E2 20751.64} C_VEL
LIN {X 0,Y 425.26,Z 297.827,A -85,B 0,C 180,E1 20749.28,E2 20749.28} C_VEL
LIN {X 0,Y 425.279,Z 297.824,A -85,B 0,C 180,E1 20745.525,E2 20745.525} C_VEL
LIN {X 0,Y 425.295,Z 297.824,A -85,B 0,C 180,E1 20741.709,E2 20741.709} C_VEL
LIN {X 0,Y 425.274,Z 297.823,A -85,B 0,C 180,E1 20738.025,E2 20738.025} C_VEL
LIN {X 0,Y 425.253,Z 297.823,A -85,B 0,C 180,E1 20734.354,E2 20734.354} C_VEL
LIN {X 0,Y 425.245,Z 297.823,A -85,B 0,C 180,E1 20730.623,E2 20730.623} C_VEL
LIN {X 0,Y 425.248,Z 297.822,A -85,B 0,C 180,E1 20726.837,E2 20726.837} C_VEL
LIN {X 0,Y 425.261,Z 297.822,A -85,B 0,C 180,E1 20723.121,E2 20723.121} C_VEL
LIN {X 0,Y 425.293,Z 297.822,A -85,B 0,C 180,E1 20719.486,E2 20719.486} C_VEL
LIN {X 0,Y 425.303,Z 297.823,A -85,B 0,C 180,E1 20715.687,E2 20715.687} C_VEL
LIN {X 0,Y 425.279,Z 297.823,A -85,B 0,C 180,E1 20711.942,E2 20711.942} C_VEL
LIN {X 0,Y 425.262,Z 297.822,A -85,B 0,C 180,E1 20708.185,E2 20708.185} C_VEL
LIN {X 0,Y 425.254,Z 297.822,A -85,B 0,C 180,E1 20704.452,E2 20704.452} C_VEL
LIN {X 0,Y 425.253,Z 297.822,A -85,B 0,C 180,E1 20700.675,E2 20700.675} C_VEL
LIN {X 0,Y 425.262,Z 297.821,A -85,B 0,C 180,E1 20696.911,E2 20696.911} C_VEL
LIN {X 0,Y 425.287,Z 297.821,A -85,B 0,C 180,E1 20693.251,E2 20693.251} C_VEL
LIN {X 0,Y 425.301,Z 297.821,A -85,B 0,C 180,E1 20689.436,E2 20689.436} C_VEL
LIN {X 0,Y 425.313,Z 297.822,A -85,B 0,C 180,E1 20685.573,E2 20685.573} C_VEL
LIN {X 0,Y 425.293,Z 297.822,A -85,B 0,C 180,E1 20681.764,E2 20681.764} C_VEL
LIN {X 0,Y 425.271,Z 297.822,A -85,B 0,C 180,E1 20678.051,E2 20678.051} C_VEL
LIN {X 0,Y 425.261,Z 297.821,A -85,B 0,C 180,E1 20674.369,E2 20674.369} C_VEL
LIN {X 0,Y 425.262,Z 297.82,A -85,B 0,C 180,E1 20670.571,E2 20670.571} C_VEL
LIN {X 0,Y 425.272,Z 297.82,A -85,B 0,C 180,E1 20666.822,E2 20666.822} C_VEL
LIN {X 0,Y 425.289,Z 297.819,A -85,B 0,C 180,E1 20663.065,E2 20663.065} C_VEL
LIN {X 0,Y 425.322,Z 297.819,A -85,B 0,C 180,E1 20659.373,E2 20659.373} C_VEL
LIN {X 0,Y 425.309,Z 297.821,A -85,B 0,C 180,E1 20655.422,E2 20655.422} C_VEL
LIN {X 0,Y 425.31,Z 297.822,A -85,B 0,C 180,E1 20651.524,E2 20651.524} C_VEL
LIN {X 0,Y 425.284,Z 297.821,A -85,B 0,C 180,E1 20647.824,E2 20647.824} C_VEL
LIN {X 0,Y 425.271,Z 297.82,A -85,B 0,C 180,E1 20644.153,E2 20644.153} C_VEL
LIN {X 0,Y 425.269,Z 297.82,A -85,B 0,C 180,E1 20640.363,E2 20640.363} C_VEL
LIN {X 0,Y 425.274,Z 297.819,A -85,B 0,C 180,E1 20636.531,E2 20636.531} C_VEL
LIN {X 0,Y 425.288,Z 297.818,A -85,B 0,C 180,E1 20632.824,E2 20632.824} C_VEL
LIN {X 0,Y 425.308,Z 297.818,A -85,B 0,C 180,E1 20629.072,E2 20629.072} C_VEL
LIN {X 0,Y 425.325,Z 297.818,A -85,B 0,C 180,E1 20625.264,E2 20625.264} C_VEL
LIN {X 0,Y 425.313,Z 297.821,A -85,B 0,C 180,E1 20621.388,E2 20621.388} C_VEL
LIN {X 0,Y 425.302,Z 297.821,A -85,B 0,C 180,E1 20617.564,E2 20617.564} C_VEL
LIN {X 0,Y 425.286,Z 297.821,A -85,B 0,C 180,E1 20613.773,E2 20613.773} C_VEL
LIN {X 0,Y 425.278,Z 297.82,A -85,B 0,C 180,E1 20609.999,E2 20609.999} C_VEL
LIN {X 0,Y 425.314,Z 297.82,A -85,B 0,C 180,E1 20607.281,E2 20607.281} C_VEL
LIN {X 0,Y 424.339,Z 297.936,A -85,B 0,C 180,E1 20606.244,E2 20606.244} C_VEL
LIN {X 0,Y 417.813,Z 298.754,A -85,B 0,C 180,E1 20603.245,E2 20603.245} C_VEL
LIN {X 0,Y 417.349,Z 298.807,A -85,B 0,C 180,E1 20602.558,E2 20602.558} C_VEL
LIN {X 0,Y 417.363,Z 298.806,A -85,B 0,C 180,E1 20598.81,E2 20598.81} C_VEL
LIN {X 0,Y 417.383,Z 298.805,A -85,B 0,C 180,E1 20595.005,E2 20595.005} C_VEL
LIN {X 0,Y 417.383,Z 298.807,A -85,B 0,C 180,E1 20591.117,E2 20591.117} C_VEL
LIN {X 0,Y 417.389,Z 298.806,A -85,B 0,C 180,E1 20587.164,E2 20587.164} C_VEL
LIN {X 0,Y 417.379,Z 298.809,A -85,B 0,C 180,E1 20583.232,E2 20583.232} C_VEL
LIN {X 0,Y 417.366,Z 298.81,A -85,B 0,C 180,E1 20579.477,E2 20579.477} C_VEL
LIN {X 0,Y 417.352,Z 298.809,A -85,B 0,C 180,E1 20575.736,E2 20575.736} C_VEL
LIN {X 0,Y 417.346,Z 298.807,A -85,B 0,C 180,E1 20571.995,E2 20571.995} C_VEL
LIN {X 0,Y 417.347,Z 298.807,A -85,B 0,C 180,E1 20568.054,E2 20568.054} C_VEL
LIN {X 0,Y 417.35,Z 298.807,A -85,B 0,C 180,E1 20564.195,E2 20564.195} C_VEL
LIN {X 0,Y 417.359,Z 298.809,A -85,B 0,C 180,E1 20560.373,E2 20560.373} C_VEL
LIN {X 0,Y 417.371,Z 298.809,A -85,B 0,C 180,E1 20556.617,E2 20556.617} C_VEL
LIN {X 0,Y 417.364,Z 298.849,A -85,B 0,C 180,E1 20555.552,E2 20555.552} C_VEL
LIN {X 0,Y 422.937,Z 318.908,A -85,B 0,C 180,E1 20551.972,E2 20551.972} C_VEL
LIN {X 0,Y 425.976,Z 331.504,A -85,B 0,C 180,E1 20549.839,E2 20549.839} C_VEL
LIN {X 0,Y 423.745,Z 359.707,A -85,B 0,C 180,E1 20545.805,E2 20545.805} C_VEL
LIN {X 0,Y 421.754,Z 388.258,A -85,B 0,C 180,E1 20541.776,E2 20541.776} C_VEL
LIN {X 0,Y 420.899,Z 403.13,A -85,B 0,C 180,E1 20539.739,E2 20539.739} C_VEL
LIN {X 0,Y 424.096,Z 426.581,A -85,B 0,C 180,E1 20539.039,E2 20539.039} C_VEL
LIN {X 0,Y 421.725,Z 526.531,A -85,B 0,C 180,E1 20536.846,E2 20536.846} C_VEL
LIN {X 0,Y 421.292,Z 542.113,A -85,B 0,C 180,E1 20536.261,E2 20536.261} C_VEL
LIN {X 0,Y 420.724,Z 557.359,A -85,B 0,C 180,E1 20535.434,E2 20535.434} C_VEL
LIN {X 0,Y 420.033,Z 572.374,A -85,B 0,C 180,E1 20534.331,E2 20534.331} C_VEL
LIN {X 0,Y 419.368,Z 585.424,A -85,B 0,C 180,E1 20533.089,E2 20533.089} C_VEL
LIN {X 0,Y 418.755,Z 597.004,A -85,B 0,C 180,E1 20531.707,E2 20531.707} C_VEL
LIN {X 0,Y 418.167,Z 608.011,A -85,B 0,C 180,E1 20530.05,E2 20530.05} C_VEL
LIN {X 0,Y 417.699,Z 617.287,A -85,B 0,C 180,E1 20528.255,E2 20528.255} C_VEL
LIN {X 0,Y 417.399,Z 624.45,A -85,B 0,C 180,E1 20526.462,E2 20526.462} C_VEL
LIN {X 0,Y 417.216,Z 630.316,A -85,B 0,C 180,E1 20524.47,E2 20524.47} C_VEL
LIN {X 0,Y 417.144,Z 634.187,A -85,B 0,C 180,E1 20522.471,E2 20522.471} C_VEL
LIN {X 0,Y 417.186,Z 636.251,A -85,B 0,C 180,E1 20520.547,E2 20520.547} C_VEL
LIN {X 0,Y 417.311,Z 636.571,A -85,B 0,C 180,E1 20518.488,E2 20518.488} C_VEL
LIN {X 0,Y 417.532,Z 635.173,A -85,B 0,C 180,E1 20516.566,E2 20516.566} C_VEL
LIN {X 0,Y 417.903,Z 631.644,A -85,B 0,C 180,E1 20514.453,E2 20514.453} C_VEL
LIN {X 0,Y 418.363,Z 626.661,A -85,B 0,C 180,E1 20512.583,E2 20512.583} C_VEL
LIN {X 0,Y 418.972,Z 620.114,A -85,B 0,C 180,E1 20510.798,E2 20510.798} C_VEL
LIN {X 0,Y 419.743,Z 611.394,A -85,B 0,C 180,E1 20509.012,E2 20509.012} C_VEL
LIN {X 0,Y 420.56,Z 602.03,A -85,B 0,C 180,E1 20507.504,E2 20507.504} C_VEL
LIN {X 0,Y 421.54,Z 589.976,A -85,B 0,C 180,E1 20505.96,E2 20505.96} C_VEL
LIN {X 0,Y 422.532,Z 576.627,A -85,B 0,C 180,E1 20504.63,E2 20504.63} C_VEL
LIN {X 0,Y 423.446,Z 562.568,A -85,B 0,C 180,E1 20503.538,E2 20503.538} C_VEL
LIN {X 0,Y 424.294,Z 547.33,A -85,B 0,C 180,E1 20502.632,E2 20502.632} C_VEL
LIN {X 0,Y 425.04,Z 530.485,A -85,B 0,C 180,E1 20501.917,E2 20501.917} C_VEL
LIN {X 0,Y 430.219,Z 441.567,A -85,B 0,C 180,E1 20499.298,E2 20499.298} C_VEL
LIN {X 0,Y 430.934,Z 428.666,A -85,B 0,C 180,E1 20498.89,E2 20498.89} C_VEL
LIN {X 0,Y 427.687,Z 409.325,A -85,B 0,C 180,E1 20497.837,E2 20497.837} C_VEL
LIN {X 0,Y 426.441,Z 402.848,A -85,B 0,C 180,E1 20497.426,E2 20497.426} C_VEL
LIN {X 0,Y 429.852,Z 377.724,A -85,B 0,C 180,E1 20493.473,E2 20493.473} C_VEL
LIN {X 0,Y 434.282,Z 353.41,A -85,B 0,C 180,E1 20489.438,E2 20489.438} C_VEL
LIN {X 0,Y 435.521,Z 347.547,A -85,B 0,C 180,E1 20488.402,E2 20488.402} C_VEL
LIN {X 0,Y 433.911,Z 339.001,A -85,B 0,C 180,E1 20486.054,E2 20486.054} C_VEL
LIN {X 0,Y 432.256,Z 332.081,A -85,B 0,C 180,E1 20483.608,E2 20483.608} C_VEL
LIN {X 0,Y 431.082,Z 328.341,A -85,B 0,C 180,E1 20481.735,E2 20481.735} C_VEL
LIN {X 0,Y 430.524,Z 326.09,A -85,B 0,C 180,E1 20480.24,E2 20480.24} C_VEL
LIN {X 0,Y 430.032,Z 324.292,A -85,B 0,C 180,E1 20477.679,E2 20477.679} C_VEL
LIN {X 0,Y 430.304,Z 324.642,A -85,B 0,C 180,E1 20475.699,E2 20475.699} C_VEL
LIN {X 0,Y 431.458,Z 327.06,A -85,B 0,C 180,E1 20473.308,E2 20473.308} C_VEL
LIN {X 0,Y 432.299,Z 329.442,A -85,B 0,C 180,E1 20472.059,E2 20472.059} C_VEL
LIN {X 0,Y 433.452,Z 332.288,A -85,B 0,C 180,E1 20470.832,E2 20470.832} C_VEL
LIN {X 0,Y 435.417,Z 337.986,A -85,B 0,C 180,E1 20468.992,E2 20468.992} C_VEL
LIN {X 0,Y 437.518,Z 345.112,A -85,B 0,C 180,E1 20467.219,E2 20467.219} C_VEL
LIN {X 0,Y 438.411,Z 349.266,A -85,B 0,C 180,E1 20466.369,E2 20466.369} C_VEL
LIN {X 0,Y 433.258,Z 374.472,A -85,B 0,C 180,E1 20463.396,E2 20463.396} C_VEL
LIN {X 0,Y 430.613,Z 392.467,A -85,B 0,C 180,E1 20461.441,E2 20461.441} C_VEL
LIN {X 0,Y 432.416,Z 409.582,A -85,B 0,C 180,E1 20460.803,E2 20460.803} C_VEL
LIN {X 0,Y 429.218,Z 505.867,A -85,B 0,C 180,E1 20458.704,E2 20458.704} C_VEL
LIN {X 0,Y 427.107,Z 586.546,A -85,B 0,C 180,E1 20457.082,E2 20457.082} C_VEL
LIN {X 0,Y 426.002,Z 606.418,A -85,B 0,C 180,E1 20456.433,E2 20456.433} C_VEL
LIN {X 0,Y 424.756,Z 624.247,A -85,B 0,C 180,E1 20455.6,E2 20455.6} C_VEL
LIN {X 0,Y 423.339,Z 642.357,A -85,B 0,C 180,E1 20454.489,E2 20454.489} C_VEL
LIN {X 0,Y 421.842,Z 659.824,A -85,B 0,C 180,E1 20453.124,E2 20453.124} C_VEL
LIN {X 0,Y 420.432,Z 675.794,A -85,B 0,C 180,E1 20451.584,E2 20451.584} C_VEL
LIN {X 0,Y 419.16,Z 691.027,A -85,B 0,C 180,E1 20449.8,E2 20449.8} C_VEL
LIN {X 0,Y 418.089,Z 704.99,A -85,B 0,C 180,E1 20447.826,E2 20447.826} C_VEL
LIN {X 0,Y 417.292,Z 717.395,A -85,B 0,C 180,E1 20445.71,E2 20445.71} C_VEL
LIN {X 0,Y 416.773,Z 728.27,A -85,B 0,C 180,E1 20443.458,E2 20443.458} C_VEL
LIN {X 0,Y 416.512,Z 737.569,A -85,B 0,C 180,E1 20441.073,E2 20441.073} C_VEL
LIN {X 0,Y 416.477,Z 744.829,A -85,B 0,C 180,E1 20438.7,E2 20438.7} C_VEL
LIN {X 0,Y 416.546,Z 750.24,A -85,B 0,C 180,E1 20436.34,E2 20436.34} C_VEL
LIN {X 0,Y 416.675,Z 753.927,A -85,B 0,C 180,E1 20433.991,E2 20433.991} C_VEL
LIN {X 0,Y 416.766,Z 755.966,A -85,B 0,C 180,E1 20431.651,E2 20431.651} C_VEL
LIN {X 0,Y 416.777,Z 756.393,A -85,B 0,C 180,E1 20429.314,E2 20429.314} C_VEL
LIN {X 0,Y 416.688,Z 755.207,A -85,B 0,C 180,E1 20426.975,E2 20426.975} C_VEL
LIN {X 0,Y 416.549,Z 752.395,A -85,B 0,C 180,E1 20424.63,E2 20424.63} C_VEL
LIN {X 0,Y 416.443,Z 747.898,A -85,B 0,C 180,E1 20422.274,E2 20422.274} C_VEL
LIN {X 0,Y 416.436,Z 741.504,A -85,B 0,C 180,E1 20419.872,E2 20419.872} C_VEL
LIN {X 0,Y 416.603,Z 733.363,A -85,B 0,C 180,E1 20417.527,E2 20417.527} C_VEL
LIN {X 0,Y 417.037,Z 723.573,A -85,B 0,C 180,E1 20415.279,E2 20415.279} C_VEL
LIN {X 0,Y 417.709,Z 712.294,A -85,B 0,C 180,E1 20413.165,E2 20413.165} C_VEL
LIN {X 0,Y 418.672,Z 699.235,A -85,B 0,C 180,E1 20411.147,E2 20411.147} C_VEL
LIN {X 0,Y 419.845,Z 684.641,A -85,B 0,C 180,E1 20409.29,E2 20409.29} C_VEL
LIN {X 0,Y 421.139,Z 669.155,A -85,B 0,C 180,E1 20407.676,E2 20407.676} C_VEL
LIN {X 0,Y 422.489,Z 652.69,A -85,B 0,C 180,E1 20406.278,E2 20406.278} C_VEL
LIN {X 0,Y 423.806,Z 635.248,A -85,B 0,C 180,E1 20405.096,E2 20405.096} C_VEL
LIN {X 0,Y 425.029,Z 616.7,A -85,B 0,C 180,E1 20404.128,E2 20404.128} C_VEL
LIN {X 0,Y 426.055,Z 598.198,A -85,B 0,C 180,E1 20403.432,E2 20403.432} C_VEL
LIN {X 0,Y 426.696,Z 579.048,A -85,B 0,C 180,E1 20402.963,E2 20402.963} C_VEL
LIN {X 0,Y 430.072,Z 412.338,A -85,B 0,C 180,E1 20399.88,E2 20399.88} C_VEL
LIN {X 0,Y 427.596,Z 388.145,A -85,B 0,C 180,E1 20399.237,E2 20399.237} C_VEL
LIN {X 0,Y 431.654,Z 345.512,A -85,B 0,C 180,E1 20395.085,E2 20395.085} C_VEL
LIN {X 0,Y 431.889,Z 340.596,A -85,B 0,C 180,E1 20394.58,E2 20394.58} C_VEL
LIN {X 0,Y 423.393,Z 315.964,A -85,B 0,C 180,E1 20391.199,E2 20391.199} C_VEL
LIN {X 0,Y 417.306,Z 298.817,A -85,B 0,C 180,E1 20388.649,E2 20388.649} C_VEL
LIN {X 0,Y 417.307,Z 298.816,A -85,B 0,C 180,E1 20384.784,E2 20384.784} C_VEL
LIN {X 0,Y 417.308,Z 298.815,A -85,B 0,C 180,E1 20381,E2 20381} C_VEL
LIN {X 0,Y 417.326,Z 298.812,A -85,B 0,C 180,E1 20377.306,E2 20377.306} C_VEL
LIN {X 0,Y 417.348,Z 298.811,A -85,B 0,C 180,E1 20373.52,E2 20373.52} C_VEL
LIN {X 0,Y 417.36,Z 298.811,A -85,B 0,C 180,E1 20369.587,E2 20369.587} C_VEL
LIN {X 0,Y 417.355,Z 298.813,A -85,B 0,C 180,E1 20365.699,E2 20365.699} C_VEL
LIN {X 0,Y 417.355,Z 298.812,A -85,B 0,C 180,E1 20361.799,E2 20361.799} C_VEL
LIN {X 0,Y 417.337,Z 298.811,A -85,B 0,C 180,E1 20357.99,E2 20357.99} C_VEL
LIN {X 0,Y 417.318,Z 298.811,A -85,B 0,C 180,E1 20354.289,E2 20354.289} C_VEL
LIN {X 0,Y 417.313,Z 298.811,A -85,B 0,C 180,E1 20350.493,E2 20350.493} C_VEL
LIN {X 0,Y 417.313,Z 298.811,A -85,B 0,C 180,E1 20346.606,E2 20346.606} C_VEL
LIN {X 0,Y 417.315,Z 298.811,A -85,B 0,C 180,E1 20342.748,E2 20342.748} C_VEL
LIN {X 0,Y 417.33,Z 298.81,A -85,B 0,C 180,E1 20339.041,E2 20339.041} C_VEL
LIN {X 0,Y 417.348,Z 298.81,A -85,B 0,C 180,E1 20335.279,E2 20335.279} C_VEL
LIN {X 0,Y 417.368,Z 298.81,A -85,B 0,C 180,E1 20331.46,E2 20331.46} C_VEL
LIN {X 0,Y 417.366,Z 298.811,A -85,B 0,C 180,E1 20327.551,E2 20327.551} C_VEL
LIN {X 0,Y 417.356,Z 298.811,A -85,B 0,C 180,E1 20323.725,E2 20323.725} C_VEL
LIN {X 0,Y 417.343,Z 298.811,A -85,B 0,C 180,E1 20319.904,E2 20319.904} C_VEL
LIN {X 0,Y 417.326,Z 298.81,A -85,B 0,C 180,E1 20316.234,E2 20316.234} C_VEL
LIN {X 0,Y 417.325,Z 298.809,A -85,B 0,C 180,E1 20312.431,E2 20312.431} C_VEL
LIN {X 0,Y 417.324,Z 298.809,A -85,B 0,C 180,E1 20308.516,E2 20308.516} C_VEL
LIN {X 0,Y 417.33,Z 298.809,A -85,B 0,C 180,E1 20304.736,E2 20304.736} C_VEL
LIN {X 0,Y 417.341,Z 298.808,A -85,B 0,C 180,E1 20300.915,E2 20300.915} C_VEL
LIN {X 0,Y 417.369,Z 298.809,A -85,B 0,C 180,E1 20297.319,E2 20297.319} C_VEL
LIN {X 0,Y 417.371,Z 298.81,A -85,B 0,C 180,E1 20293.434,E2 20293.434} C_VEL
LIN {X 0,Y 417.374,Z 298.811,A -85,B 0,C 180,E1 20289.527,E2 20289.527} C_VEL
LIN {X 0,Y 417.361,Z 298.811,A -85,B 0,C 180,E1 20285.6,E2 20285.6} C_VEL
LIN {X 0,Y 417.348,Z 298.81,A -85,B 0,C 180,E1 20281.806,E2 20281.806} C_VEL
LIN {X 0,Y 417.334,Z 298.809,A -85,B 0,C 180,E1 20278.161,E2 20278.161} C_VEL
LIN {X 0,Y 417.333,Z 298.808,A -85,B 0,C 180,E1 20274.334,E2 20274.334} C_VEL
LIN {X 0,Y 417.335,Z 298.808,A -85,B 0,C 180,E1 20270.473,E2 20270.473} C_VEL
LIN {X 0,Y 417.344,Z 298.807,A -85,B 0,C 180,E1 20266.707,E2 20266.707} C_VEL
LIN {X 0,Y 417.367,Z 298.807,A -85,B 0,C 180,E1 20263.013,E2 20263.013} C_VEL
LIN {X 0,Y 417.375,Z 298.807,A -85,B 0,C 180,E1 20259.096,E2 20259.096} C_VEL
LIN {X 0,Y 417.378,Z 298.808,A -85,B 0,C 180,E1 20255.222,E2 20255.222} C_VEL
LIN {X 0,Y 417.381,Z 298.808,A -85,B 0,C 180,E1 20251.234,E2 20251.234} C_VEL
LIN {X 0,Y 417.375,Z 298.81,A -85,B 0,C 180,E1 20247.317,E2 20247.317} C_VEL
LIN {X 0,Y 417.375,Z 298.811,A -85,B 0,C 180,E1 20243.396,E2 20243.396} C_VEL
LIN {X 0,Y 417.349,Z 298.807,A -85,B 0,C 180,E1 20242.558,E2 20242.558} C_VEL
LIN {X 0,Y 416.317,Z 298.942,A -85,B 0,C 180,E1 20241.5,E2 20241.5} C_VEL
LIN {X 0,Y 409.812,Z 299.747,A -85,B 0,C 180,E1 20238.442,E2 20238.442} C_VEL
LIN {X 0,Y 409.412,Z 299.798,A -85,B 0,C 180,E1 20237.741,E2 20237.741} C_VEL
LIN {X 0,Y 409.404,Z 299.797,A -85,B 0,C 180,E1 20233.979,E2 20233.979} C_VEL
LIN {X 0,Y 409.403,Z 299.797,A -85,B 0,C 180,E1 20230.086,E2 20230.086} C_VEL
LIN {X 0,Y 409.407,Z 299.796,A -85,B 0,C 180,E1 20226.235,E2 20226.235} C_VEL
LIN {X 0,Y 409.411,Z 299.795,A -85,B 0,C 180,E1 20222.352,E2 20222.352} C_VEL
LIN {X 0,Y 409.417,Z 299.795,A -85,B 0,C 180,E1 20218.491,E2 20218.491} C_VEL
LIN {X 0,Y 409.424,Z 299.794,A -85,B 0,C 180,E1 20214.634,E2 20214.634} C_VEL
LIN {X 0,Y 409.436,Z 299.793,A -85,B 0,C 180,E1 20210.721,E2 20210.721} C_VEL
LIN {X 0,Y 409.439,Z 299.794,A -85,B 0,C 180,E1 20206.86,E2 20206.86} C_VEL
LIN {X 0,Y 409.442,Z 299.798,A -85,B 0,C 180,E1 20202.894,E2 20202.894} C_VEL
LIN {X 0,Y 409.451,Z 299.797,A -85,B 0,C 180,E1 20199.048,E2 20199.048} C_VEL
